(* CODESYS project SLL_IFM_IO_V0.0.1.0_SP16p5.library
   Version: 0.0.1.0
   Title: SLL_IFM_IO
   Placeholder: SLL_IFM_IO
   CompiledLibraryCompatibilityVersion: CODESYS V3.5 SP16 Patch 5
   Company: SLL
   DefaultNamespace: SLL_IFM_IO

Project tree, tasks and I/O mapping:
  libraries: Util, 3.5.15.0 (System); Standard, 3.5.15.0 (System); ifmIOcommon, 2.4.0.0 (ifm electronic); ifmIOconfigDiagProt, 2.0.6.0 (ifm electronic); ifmTypes, 1.9.6.0 (ifm electronic); BASIC, 3.3.3.0 (OSCAT); ifmOutGroup, 2.1.3.0 (ifm electronic); ifmRawCAN, 4.0.3.0 (ifm electronic); ifmDeviceCR07nn, 1.2.2.0 (ifm electronic); SLL_IFM_Version, 0.0.0.2 (SLL)
  Library Information/
    function IsLibReleased [ST]
    function GetLibVersionNumber [ST]
    function GetLibVersion [ST]
  IO/
    data type CRXXXX_OUTPUT_GROUP_PINS
    data type CRXXXX_INPUT_PINS
    CR0709/
      data type CR0709_ALL_INPUTS_DATA
      data type CR0709_ALL_INPUTS_FB
      data type CR0709_ALL_OUTPUTS_DATA
      data type CR0709_ALL_OUTPUTS_FB
      data type CR0709_ALL_OUTPUT_STATES
      Output/
        function CR0709_Get_Output_Pin_Name_Str [ST]
        function CR0709_Get_Output_Pin_Number_Str [ST]
        function CR0709_Get_Output_Pin_Group [ST]
      Input/
        function CR0709_Get_Input_Pin_Number_Str [ST]
        function CR0709_Get_Input_Pin_Name_Str [ST]
      program PLC_CR0709_System [FBD]
    CR721S/
      data type CR721S_ALL_INPUTS_DATA
      data type CR721S_ALL_INPUTS_FB
      data type CR721S_ALL_OUTPUTS_DATA
      data type CR721S_ALL_OUTPUTS_FB
      data type CR721S_ALL_OUTPUT_STATES
    data type CRXXXX_INPUT_DATA
    data type CRXXXX_OUTPUT_DATA
    data type CRXXXX_OUTPUT_STATE_DATA
    FB/
      function block CRXXXX_INPUT_FB [FBD]: Process
      function block CRXXXX_OUTPUT_FB [FBD]: Process
      function block CRXXXX_OUTPUT_GROUP_FB [FBD]: Process
    Input/
      function CR721S_Get_Input_Pin_Number_Str [ST]
      function CR721S_Get_Input_Pin_Name_Str [ST]
      function CR721S_Get_Input_Pin_Connector [ST]
    Output/
      function CR721S_Get_Output_Group_Pin_Number_Str [ST]
      function CR721S_Get_Output_Group_Pin_Name_Str [ST]
      function CR721S_Get_Output_Pin_Name_Str [ST]
      function CR721S_Get_Output_Pin_Number_Str [ST]
      function CR721S_Get_Output_Pin_Group [ST]
      function CR721S_Get_Output_Pin_Connector [ST]
    data type CRXXXX_OUTPUT_PINS
    data type CRXXXX_OUTPUT_GROUP_DATA
    data type CRXXXX_VERSION_DATA
  global variables GVL_IfmIoLibs
  Hardware/
    data type CRXXXX_LINAK_STATUS
    function block Diag_Op_LINAK_Bridge [FBD]
    data type Diag_Op_PWM_Enum
    data type CRXXXX_Freq_Pulse_Readings
    data type Diag_Ip_Signal_Enum
  Func/
    function Get_IFM_DIAG_INFO_STRING [ST]
*)

// IO/CRXXXX_OUTPUT_GROUP_PINS
{attribute 'qualified_only'}
//{attribute 'strict'}
{attribute 'to_string'} 
TYPE CRXXXX_OUTPUT_GROUP_PINS :
(
	GROUP0 :=0000,
	GROUP1 :=0001,
	GROUP2 :=0002,
	GROUP3 :=0003,
	GROUP4 :=0004,
	GROUP5 :=0005
)WORD;
END_TYPE

// IO/CR0709/CR0709_ALL_INPUTS_DATA
TYPE CR0709_ALL_INPUTS_DATA :
STRUCT
	VERSION: DWORD:=16#8000001;	
	IN0100: CRXXXX_INPUT_DATA;
	IN0101: CRXXXX_INPUT_DATA;
	IN0102: CRXXXX_INPUT_DATA;
	IN0103: CRXXXX_INPUT_DATA;
	IN0200: CRXXXX_INPUT_DATA;
	IN0201: CRXXXX_INPUT_DATA;
	IN0202: CRXXXX_INPUT_DATA;
	IN0203: CRXXXX_INPUT_DATA;
	IN0600: CRXXXX_INPUT_DATA;
	IN0601: CRXXXX_INPUT_DATA;
	IN0602: CRXXXX_INPUT_DATA;
	IN0603: CRXXXX_INPUT_DATA;
	IN0700: CRXXXX_INPUT_DATA;
	IN0701: CRXXXX_INPUT_DATA;
	IN0702: CRXXXX_INPUT_DATA;
	IN0703: CRXXXX_INPUT_DATA;
	IN0000: CRXXXX_INPUT_DATA;
	IN0001: CRXXXX_INPUT_DATA;
	IN0002: CRXXXX_INPUT_DATA;
	IN0003: CRXXXX_INPUT_DATA;
	IN0500: CRXXXX_INPUT_DATA;
	IN0501: CRXXXX_INPUT_DATA;
	IN0502: CRXXXX_INPUT_DATA;
	IN0503: CRXXXX_INPUT_DATA;
	IN0400: CRXXXX_INPUT_DATA;
	IN0401: CRXXXX_INPUT_DATA;
	IN0900: CRXXXX_INPUT_DATA;
	IN0901: CRXXXX_INPUT_DATA;
	IN0300: CRXXXX_INPUT_DATA;
	IN0301: CRXXXX_INPUT_DATA;
	IN0800: CRXXXX_INPUT_DATA;
	IN0801: CRXXXX_INPUT_DATA;
END_STRUCT
END_TYPE

// IO/CR0709/CR0709_ALL_INPUTS_FB
TYPE CR0709_ALL_INPUTS_FB :
STRUCT
	VERSION: DWORD:=16#8000001;	
	IN0100: CRXXXX_INPUT_FB;
	IN0101: CRXXXX_INPUT_FB;
	IN0102: CRXXXX_INPUT_FB;
	IN0103: CRXXXX_INPUT_FB;
	IN0200: CRXXXX_INPUT_FB;
	IN0201: CRXXXX_INPUT_FB;
	IN0202: CRXXXX_INPUT_FB;
	IN0203: CRXXXX_INPUT_FB;
	IN0600: CRXXXX_INPUT_FB;
	IN0601: CRXXXX_INPUT_FB;
	IN0602: CRXXXX_INPUT_FB;
	IN0603: CRXXXX_INPUT_FB;
	IN0700: CRXXXX_INPUT_FB;
	IN0701: CRXXXX_INPUT_FB;
	IN0702: CRXXXX_INPUT_FB;
	IN0703: CRXXXX_INPUT_FB;
	IN0000: CRXXXX_INPUT_FB;
	IN0001: CRXXXX_INPUT_FB;
	IN0002: CRXXXX_INPUT_FB;
	IN0003: CRXXXX_INPUT_FB;
	IN0500: CRXXXX_INPUT_FB;
	IN0501: CRXXXX_INPUT_FB;
	IN0502: CRXXXX_INPUT_FB;
	IN0503: CRXXXX_INPUT_FB;
	IN0400: CRXXXX_INPUT_FB;
	IN0401: CRXXXX_INPUT_FB;
	IN0900: CRXXXX_INPUT_FB;
	IN0901: CRXXXX_INPUT_FB;
	IN0300: CRXXXX_INPUT_FB;
	IN0301: CRXXXX_INPUT_FB;
	IN0800: CRXXXX_INPUT_FB;
	IN0801: CRXXXX_INPUT_FB;	
END_STRUCT
END_TYPE

// IO/CRXXXX_INPUT_PINS
{attribute 'qualified_only'}
//{attribute 'strict'}
{attribute 'to_string'}
TYPE CRXXXX_INPUT_PINS :
(
	IN0100:=0100,
	IN0101:=0101,
	IN0102:=0102,
	IN0103:=0103,
	IN0200:=0200,
	IN0201:=0201,
	IN0202:=0202,
	IN0203:=0203,
	IN0600:=0600,
	IN0601:=0601,
	IN0602:=0602,
	IN0603:=0603,
	IN0700:=0700,
	IN0701:=0701,
	IN0702:=0702,
	IN0703:=0703,
	IN0000:=0000,
	IN0001:=0001,
	IN0002:=0002,
	IN0003:=0003,
	IN0500:=0500,
	IN0501:=0501,
	IN0502:=0502,
	IN0503:=0503,
	IN0400:=0400,
	IN0401:=0401,
	IN0900:=0900,
	IN0901:=0901,
	IN0300:=0300,
	IN0301:=0301,
	IN0800:=0800,
	IN0801:=0801,
	
	IN1100:=1100,
	IN1101:=1101,
	IN1102:=1102,
	IN1103:=1103,
	IN1600:=1600,
	IN1601:=1601,
	IN1602:=1602,
	IN1603:=1603,
	
	IN1000:=1000,
	IN1001:=1001,
	IN1002:=1002,
	IN1003:=1003,
	IN1500:=1500,
	IN1501:=1501,
	IN1502:=1502,
	IN1503:=1503,

	IN1200:=1200,
	IN1201:=1201,
	IN1202:=1202,
	IN1203:=1203,
	IN1400:=1400,
	IN1401:=1401,
	IN1402:=1402,
	IN1403:=1403,
	IN1700:=1700,
	IN1701:=1701,
	IN1702:=1702,
	IN1703:=1703,
	IN1800:=1800,
	IN1801:=1801,
	IN1802:=1802,
	IN1803:=1803,
	IN1300:=1300,
	IN1301:=1301,
	IN1302:=1302,
	IN1303:=1303
)WORD;
END_TYPE;

// IO/CR0709/CR0709_ALL_OUTPUTS_DATA
TYPE CR0709_ALL_OUTPUTS_DATA :
STRUCT
	VERSION: DWORD:=16#8000001;	
	OUT0000 : CRXXXX_OUTPUT_DATA;
	OUT0001 : CRXXXX_OUTPUT_DATA;
	OUT0002 : CRXXXX_OUTPUT_DATA;
	OUT0003 : CRXXXX_OUTPUT_DATA;
	OUT0004 : CRXXXX_OUTPUT_DATA;
	OUT0005 : CRXXXX_OUTPUT_DATA;
	OUT0006 : CRXXXX_OUTPUT_DATA;
	OUT0007 : CRXXXX_OUTPUT_DATA;
	OUT0008 : CRXXXX_OUTPUT_DATA;
	OUT0100 : CRXXXX_OUTPUT_DATA;
	OUT0101 : CRXXXX_OUTPUT_DATA;
	OUT0102 : CRXXXX_OUTPUT_DATA;
	OUT0103 : CRXXXX_OUTPUT_DATA;
	OUT0104 : CRXXXX_OUTPUT_DATA;
	OUT0105 : CRXXXX_OUTPUT_DATA;
	OUT0106 : CRXXXX_OUTPUT_DATA;
	OUT0107 : CRXXXX_OUTPUT_DATA;
	OUT0108 : CRXXXX_OUTPUT_DATA;
	OUT0200 : CRXXXX_OUTPUT_DATA;
	OUT0201 : CRXXXX_OUTPUT_DATA;
	OUT0202 : CRXXXX_OUTPUT_DATA;
	OUT0203 : CRXXXX_OUTPUT_DATA;
	OUT0204 : CRXXXX_OUTPUT_DATA;
	OUT0205 : CRXXXX_OUTPUT_DATA;
	OUT0206 : CRXXXX_OUTPUT_DATA;
	OUT0207 : CRXXXX_OUTPUT_DATA;
	OUT0208 : CRXXXX_OUTPUT_DATA;
	OUT3000 : CRXXXX_OUTPUT_DATA;
	OUT3001 : CRXXXX_OUTPUT_DATA;
	
	GROUP0 : CRXXXX_OUTPUT_GROUP_DATA;
	GROUP1 : CRXXXX_OUTPUT_GROUP_DATA;
	GROUP2 : CRXXXX_OUTPUT_GROUP_DATA;
END_STRUCT
END_TYPE

// IO/CR0709/CR0709_ALL_OUTPUTS_FB
TYPE CR0709_ALL_OUTPUTS_FB :
STRUCT
	VERSION: DWORD:=16#8000001;	
	OUT0000 : CRXXXX_OUTPUT_FB;
	OUT0001 : CRXXXX_OUTPUT_FB;
	OUT0002 : CRXXXX_OUTPUT_FB;
	OUT0003 : CRXXXX_OUTPUT_FB;
	OUT0004 : CRXXXX_OUTPUT_FB;
	OUT0005 : CRXXXX_OUTPUT_FB;
	OUT0006 : CRXXXX_OUTPUT_FB;
	OUT0007 : CRXXXX_OUTPUT_FB;
	OUT0008 : CRXXXX_OUTPUT_FB;
	OUT0100 : CRXXXX_OUTPUT_FB;
	OUT0101 : CRXXXX_OUTPUT_FB;
	OUT0102 : CRXXXX_OUTPUT_FB;
	OUT0103 : CRXXXX_OUTPUT_FB;
	OUT0104 : CRXXXX_OUTPUT_FB;
	OUT0105 : CRXXXX_OUTPUT_FB;
	OUT0106 : CRXXXX_OUTPUT_FB;
	OUT0107 : CRXXXX_OUTPUT_FB;
	OUT0108 : CRXXXX_OUTPUT_FB;
	OUT0200 : CRXXXX_OUTPUT_FB;
	OUT0201 : CRXXXX_OUTPUT_FB;
	OUT0202 : CRXXXX_OUTPUT_FB;
	OUT0203 : CRXXXX_OUTPUT_FB;
	OUT0204 : CRXXXX_OUTPUT_FB;
	OUT0205 : CRXXXX_OUTPUT_FB;
	OUT0206 : CRXXXX_OUTPUT_FB;
	OUT0207 : CRXXXX_OUTPUT_FB;
	OUT0208 : CRXXXX_OUTPUT_FB;
	OUT3000 : CRXXXX_OUTPUT_FB;
	OUT3001 : CRXXXX_OUTPUT_FB;
	
	GROUP0 : CRXXXX_OUTPUT_GROUP_FB;
	GROUP1 : CRXXXX_OUTPUT_GROUP_FB;
	GROUP2 : CRXXXX_OUTPUT_GROUP_FB;	
END_STRUCT
END_TYPE

// IO/CR0709/CR0709_ALL_OUTPUT_STATES
TYPE CR0709_ALL_OUTPUT_STATES :
STRUCT
	VERSION: DWORD:=16#8000001;	
	OUT0000 : CRXXXX_OUTPUT_STATE_DATA;
	OUT0001 : CRXXXX_OUTPUT_STATE_DATA;
	OUT0002 : CRXXXX_OUTPUT_STATE_DATA;
	OUT0003 : CRXXXX_OUTPUT_STATE_DATA;
	OUT0004 : CRXXXX_OUTPUT_STATE_DATA;
	OUT0005 : CRXXXX_OUTPUT_STATE_DATA;
	OUT0006 : CRXXXX_OUTPUT_STATE_DATA;
	OUT0007 : CRXXXX_OUTPUT_STATE_DATA;
	OUT0008 : CRXXXX_OUTPUT_STATE_DATA;
	OUT0100 : CRXXXX_OUTPUT_STATE_DATA;
	OUT0101 : CRXXXX_OUTPUT_STATE_DATA;
	OUT0102 : CRXXXX_OUTPUT_STATE_DATA;
	OUT0103 : CRXXXX_OUTPUT_STATE_DATA;
	OUT0104 : CRXXXX_OUTPUT_STATE_DATA;
	OUT0105 : CRXXXX_OUTPUT_STATE_DATA;
	OUT0106 : CRXXXX_OUTPUT_STATE_DATA;
	OUT0107 : CRXXXX_OUTPUT_STATE_DATA;
	OUT0108 : CRXXXX_OUTPUT_STATE_DATA;
	OUT0200 : CRXXXX_OUTPUT_STATE_DATA;
	OUT0201 : CRXXXX_OUTPUT_STATE_DATA;
	OUT0202 : CRXXXX_OUTPUT_STATE_DATA;
	OUT0203 : CRXXXX_OUTPUT_STATE_DATA;
	OUT0204 : CRXXXX_OUTPUT_STATE_DATA;
	OUT0205 : CRXXXX_OUTPUT_STATE_DATA;
	OUT0206 : CRXXXX_OUTPUT_STATE_DATA;
	OUT0207 : CRXXXX_OUTPUT_STATE_DATA;
	OUT0208 : CRXXXX_OUTPUT_STATE_DATA;
	OUT3000 : CRXXXX_OUTPUT_STATE_DATA;
	OUT3001 : CRXXXX_OUTPUT_STATE_DATA;
	
	GROUP0: CRXXXX_OUTPUT_STATE_DATA;
	GROUP1: CRXXXX_OUTPUT_STATE_DATA;
	GROUP2: CRXXXX_OUTPUT_STATE_DATA;	
END_STRUCT
END_TYPE

// IO/CRXXXX_INPUT_DATA
TYPE CRXXXX_INPUT_DATA :
STRUCT
	uiChannel:WORD;
	eMode: ifmIOcommon.MODE_INPUT;
	eFilter: ifmIOcommon.FILTER_INPUT;

	xError:BOOL;
	eDiagInfo:ifmTypes.DIAG_INFO;
	xPrepared:BOOL;
	xValueDigital:BOOL;
	xValueDigital_Prev:BOOL;	
	uiValueAnalogue:UINT;	
	DigitalChanges:WORD;
	
	Signal_Type: Diag_Ip_Signal_Enum;
END_STRUCT
END_TYPE

// IO/CR721S/CR721S_ALL_INPUTS_DATA
TYPE CR721S_ALL_INPUTS_DATA :
STRUCT
	VERSION: DWORD:=16#8000001;	
	IN0100: CRXXXX_INPUT_DATA;
	IN0101: CRXXXX_INPUT_DATA;
	IN0102: CRXXXX_INPUT_DATA;
	IN0103: CRXXXX_INPUT_DATA;
	IN0200: CRXXXX_INPUT_DATA;
	IN0201: CRXXXX_INPUT_DATA;
	IN0202: CRXXXX_INPUT_DATA;
	IN0203: CRXXXX_INPUT_DATA;
	IN0600: CRXXXX_INPUT_DATA;
	IN0601: CRXXXX_INPUT_DATA;
	IN0602: CRXXXX_INPUT_DATA;
	IN0603: CRXXXX_INPUT_DATA;
	IN0700: CRXXXX_INPUT_DATA;
	IN0701: CRXXXX_INPUT_DATA;
	IN0702: CRXXXX_INPUT_DATA;
	IN0703: CRXXXX_INPUT_DATA;
	IN0000: CRXXXX_INPUT_DATA;
	IN0001: CRXXXX_INPUT_DATA;
	IN0002: CRXXXX_INPUT_DATA;
	IN0003: CRXXXX_INPUT_DATA;
	IN0500: CRXXXX_INPUT_DATA;
	IN0501: CRXXXX_INPUT_DATA;
	IN0502: CRXXXX_INPUT_DATA;
	IN0503: CRXXXX_INPUT_DATA;
	IN0400: CRXXXX_INPUT_DATA;
	IN0401: CRXXXX_INPUT_DATA;
	IN0900: CRXXXX_INPUT_DATA;
	IN0901: CRXXXX_INPUT_DATA;
	IN0300: CRXXXX_INPUT_DATA;
	IN0301: CRXXXX_INPUT_DATA;
	IN0800: CRXXXX_INPUT_DATA;
	IN0801: CRXXXX_INPUT_DATA;
	
	IN1100: CRXXXX_INPUT_DATA;
	IN1101: CRXXXX_INPUT_DATA;
	IN1102: CRXXXX_INPUT_DATA;
	IN1103: CRXXXX_INPUT_DATA;
	IN1600: CRXXXX_INPUT_DATA;
	IN1601: CRXXXX_INPUT_DATA;
	IN1602: CRXXXX_INPUT_DATA;
	IN1603: CRXXXX_INPUT_DATA;
	
	IN1000: CRXXXX_INPUT_DATA;
	IN1001: CRXXXX_INPUT_DATA;
	IN1002: CRXXXX_INPUT_DATA;
	IN1003: CRXXXX_INPUT_DATA;
	IN1500: CRXXXX_INPUT_DATA;
	IN1501: CRXXXX_INPUT_DATA;
	IN1502: CRXXXX_INPUT_DATA;
	IN1503: CRXXXX_INPUT_DATA;

	IN1200: CRXXXX_INPUT_DATA;
	IN1201: CRXXXX_INPUT_DATA;
	IN1202: CRXXXX_INPUT_DATA;
	IN1203: CRXXXX_INPUT_DATA;
	IN1400: CRXXXX_INPUT_DATA;
	IN1401: CRXXXX_INPUT_DATA;
	IN1402: CRXXXX_INPUT_DATA;
	IN1403: CRXXXX_INPUT_DATA;
	IN1700: CRXXXX_INPUT_DATA;
	IN1701: CRXXXX_INPUT_DATA;
	IN1702: CRXXXX_INPUT_DATA;
	IN1703: CRXXXX_INPUT_DATA;
	IN1800: CRXXXX_INPUT_DATA;
	IN1801: CRXXXX_INPUT_DATA;
	IN1802: CRXXXX_INPUT_DATA;
	IN1803: CRXXXX_INPUT_DATA;
	IN1300: CRXXXX_INPUT_DATA;
	IN1301: CRXXXX_INPUT_DATA;
	IN1302: CRXXXX_INPUT_DATA;
	IN1303: CRXXXX_INPUT_DATA;
END_STRUCT
END_TYPE

// IO/CRXXXX_OUTPUT_DATA
TYPE CRXXXX_OUTPUT_DATA :
STRUCT
	uiChannel:WORD;
	eMode: ifmIOcommon.MODE_OUTPUT;
	eFilter: ifmIOcommon.FILTER_OUTPUT;	
	uiOpValue: UINT;
	PWM_Flags: Diag_Op_PWM_Enum;
	
	xError:BOOL;
	eDiagInfo:ifmTypes.DIAG_INFO;	
	xPrepared:BOOL;
	xOutState:BOOL;
	uiOutVoltage:UINT;
	uiOutCurrent:UINT;
	
	xGroupError:BOOL;
	xGroupPrepared:BOOL;
	xGroupGroupState:BOOL;
	xGroupValue:BOOL;
END_STRUCT
END_TYPE

// IO/CRXXXX_OUTPUT_STATE_DATA
TYPE CRXXXX_OUTPUT_STATE_DATA :
STRUCT
	uiValue: UINT;
	xReset: BOOL;
	xManAuto: BOOL;
	uiManValue: UINT;
END_STRUCT
END_TYPE

// IO/CR721S/CR721S_ALL_INPUTS_FB
TYPE CR721S_ALL_INPUTS_FB :
STRUCT
	VERSION: DWORD:=16#8000001;	
	IN0100: CRXXXX_INPUT_FB;
	IN0101: CRXXXX_INPUT_FB;
	IN0102: CRXXXX_INPUT_FB;
	IN0103: CRXXXX_INPUT_FB;
	IN0200: CRXXXX_INPUT_FB;
	IN0201: CRXXXX_INPUT_FB;
	IN0202: CRXXXX_INPUT_FB;
	IN0203: CRXXXX_INPUT_FB;
	IN0600: CRXXXX_INPUT_FB;
	IN0601: CRXXXX_INPUT_FB;
	IN0602: CRXXXX_INPUT_FB;
	IN0603: CRXXXX_INPUT_FB;
	IN0700: CRXXXX_INPUT_FB;
	IN0701: CRXXXX_INPUT_FB;
	IN0702: CRXXXX_INPUT_FB;
	IN0703: CRXXXX_INPUT_FB;
	IN0000: CRXXXX_INPUT_FB;
	IN0001: CRXXXX_INPUT_FB;
	IN0002: CRXXXX_INPUT_FB;
	IN0003: CRXXXX_INPUT_FB;
	IN0500: CRXXXX_INPUT_FB;
	IN0501: CRXXXX_INPUT_FB;
	IN0502: CRXXXX_INPUT_FB;
	IN0503: CRXXXX_INPUT_FB;
	IN0400: CRXXXX_INPUT_FB;
	IN0401: CRXXXX_INPUT_FB;
	IN0900: CRXXXX_INPUT_FB;
	IN0901: CRXXXX_INPUT_FB;
	IN0300: CRXXXX_INPUT_FB;
	IN0301: CRXXXX_INPUT_FB;
	IN0800: CRXXXX_INPUT_FB;
	IN0801: CRXXXX_INPUT_FB;
	
	IN1100: CRXXXX_INPUT_FB;
	IN1101: CRXXXX_INPUT_FB;
	IN1102: CRXXXX_INPUT_FB;
	IN1103: CRXXXX_INPUT_FB;
	IN1600: CRXXXX_INPUT_FB;
	IN1601: CRXXXX_INPUT_FB;
	IN1602: CRXXXX_INPUT_FB;
	IN1603: CRXXXX_INPUT_FB;
	
	IN1000: CRXXXX_INPUT_FB;
	IN1001: CRXXXX_INPUT_FB;
	IN1002: CRXXXX_INPUT_FB;
	IN1003: CRXXXX_INPUT_FB;
	IN1500: CRXXXX_INPUT_FB;
	IN1501: CRXXXX_INPUT_FB;
	IN1502: CRXXXX_INPUT_FB;
	IN1503: CRXXXX_INPUT_FB;

	IN1200: CRXXXX_INPUT_FB;
	IN1201: CRXXXX_INPUT_FB;
	IN1202: CRXXXX_INPUT_FB;
	IN1203: CRXXXX_INPUT_FB;
	IN1400: CRXXXX_INPUT_FB;
	IN1401: CRXXXX_INPUT_FB;
	IN1402: CRXXXX_INPUT_FB;
	IN1403: CRXXXX_INPUT_FB;
	IN1700: CRXXXX_INPUT_FB;
	IN1701: CRXXXX_INPUT_FB;
	IN1702: CRXXXX_INPUT_FB;
	IN1703: CRXXXX_INPUT_FB;
	IN1800: CRXXXX_INPUT_FB;
	IN1801: CRXXXX_INPUT_FB;
	IN1802: CRXXXX_INPUT_FB;
	IN1803: CRXXXX_INPUT_FB;
	IN1300: CRXXXX_INPUT_FB;
	IN1301: CRXXXX_INPUT_FB;
	IN1302: CRXXXX_INPUT_FB;
	IN1303: CRXXXX_INPUT_FB;
END_STRUCT
END_TYPE

// IO/CR721S/CR721S_ALL_OUTPUTS_DATA
TYPE CR721S_ALL_OUTPUTS_DATA :
STRUCT
	VERSION: DWORD:=16#8000001;	
	OUT0000 : CRXXXX_OUTPUT_DATA;
	OUT0001 : CRXXXX_OUTPUT_DATA;
	OUT0002 : CRXXXX_OUTPUT_DATA;
	OUT0003 : CRXXXX_OUTPUT_DATA;
	OUT0004 : CRXXXX_OUTPUT_DATA;
	OUT0005 : CRXXXX_OUTPUT_DATA;
	OUT0006 : CRXXXX_OUTPUT_DATA;
	OUT0007 : CRXXXX_OUTPUT_DATA;
	OUT0008 : CRXXXX_OUTPUT_DATA;
	OUT0100 : CRXXXX_OUTPUT_DATA;
	OUT0101 : CRXXXX_OUTPUT_DATA;
	OUT0102 : CRXXXX_OUTPUT_DATA;
	OUT0103 : CRXXXX_OUTPUT_DATA;
	OUT0104 : CRXXXX_OUTPUT_DATA;
	OUT0105 : CRXXXX_OUTPUT_DATA;
	OUT0106 : CRXXXX_OUTPUT_DATA;
	OUT0107 : CRXXXX_OUTPUT_DATA;
	OUT0108 : CRXXXX_OUTPUT_DATA;
	OUT0200 : CRXXXX_OUTPUT_DATA;
	OUT0201 : CRXXXX_OUTPUT_DATA;
	OUT0202 : CRXXXX_OUTPUT_DATA;
	OUT0203 : CRXXXX_OUTPUT_DATA;
	OUT0204 : CRXXXX_OUTPUT_DATA;
	OUT0205 : CRXXXX_OUTPUT_DATA;
	OUT0206 : CRXXXX_OUTPUT_DATA;
	OUT0207 : CRXXXX_OUTPUT_DATA;
	OUT0208 : CRXXXX_OUTPUT_DATA;
	OUT3000 : CRXXXX_OUTPUT_DATA;
	OUT3001 : CRXXXX_OUTPUT_DATA;
	
	OUT0300 : CRXXXX_OUTPUT_DATA;
	OUT0301 : CRXXXX_OUTPUT_DATA;
	OUT0302 : CRXXXX_OUTPUT_DATA;
	OUT0303 : CRXXXX_OUTPUT_DATA;
	OUT0304 : CRXXXX_OUTPUT_DATA;
	OUT0305 : CRXXXX_OUTPUT_DATA;
	OUT0306 : CRXXXX_OUTPUT_DATA;
	OUT0307 : CRXXXX_OUTPUT_DATA;
	OUT0308 : CRXXXX_OUTPUT_DATA;
	OUT0400 : CRXXXX_OUTPUT_DATA;
	OUT0401 : CRXXXX_OUTPUT_DATA;
	OUT0402 : CRXXXX_OUTPUT_DATA;
	OUT0403 : CRXXXX_OUTPUT_DATA;
	OUT0404 : CRXXXX_OUTPUT_DATA;
	OUT0405 : CRXXXX_OUTPUT_DATA;
	OUT0406 : CRXXXX_OUTPUT_DATA;
	OUT0407 : CRXXXX_OUTPUT_DATA;
	OUT0408 : CRXXXX_OUTPUT_DATA;
	OUT0500 : CRXXXX_OUTPUT_DATA;
	OUT0501 : CRXXXX_OUTPUT_DATA;
	OUT0502 : CRXXXX_OUTPUT_DATA;
	OUT0503 : CRXXXX_OUTPUT_DATA;
	OUT0504 : CRXXXX_OUTPUT_DATA;
	OUT0505 : CRXXXX_OUTPUT_DATA;
	OUT0506 : CRXXXX_OUTPUT_DATA;
	OUT0507 : CRXXXX_OUTPUT_DATA;
	OUT0508 : CRXXXX_OUTPUT_DATA;
	OUT3002 : CRXXXX_OUTPUT_DATA;
	
	GROUP0 : CRXXXX_OUTPUT_GROUP_DATA;
	GROUP1 : CRXXXX_OUTPUT_GROUP_DATA;
	GROUP2 : CRXXXX_OUTPUT_GROUP_DATA;
	GROUP3 : CRXXXX_OUTPUT_GROUP_DATA;
	GROUP4 : CRXXXX_OUTPUT_GROUP_DATA;
	GROUP5 : CRXXXX_OUTPUT_GROUP_DATA;	
END_STRUCT
END_TYPE

// IO/CR721S/CR721S_ALL_OUTPUTS_FB
TYPE CR721S_ALL_OUTPUTS_FB :
STRUCT
	VERSION: DWORD:=16#8000001;	
	OUT0000 : CRXXXX_OUTPUT_FB;
	OUT0001 : CRXXXX_OUTPUT_FB;
	OUT0002 : CRXXXX_OUTPUT_FB;
	OUT0003 : CRXXXX_OUTPUT_FB;
	OUT0004 : CRXXXX_OUTPUT_FB;
	OUT0005 : CRXXXX_OUTPUT_FB;
	OUT0006 : CRXXXX_OUTPUT_FB;
	OUT0007 : CRXXXX_OUTPUT_FB;
	OUT0008 : CRXXXX_OUTPUT_FB;
	OUT0100 : CRXXXX_OUTPUT_FB;
	OUT0101 : CRXXXX_OUTPUT_FB;
	OUT0102 : CRXXXX_OUTPUT_FB;
	OUT0103 : CRXXXX_OUTPUT_FB;
	OUT0104 : CRXXXX_OUTPUT_FB;
	OUT0105 : CRXXXX_OUTPUT_FB;
	OUT0106 : CRXXXX_OUTPUT_FB;
	OUT0107 : CRXXXX_OUTPUT_FB;
	OUT0108 : CRXXXX_OUTPUT_FB;
	OUT0200 : CRXXXX_OUTPUT_FB;
	OUT0201 : CRXXXX_OUTPUT_FB;
	OUT0202 : CRXXXX_OUTPUT_FB;
	OUT0203 : CRXXXX_OUTPUT_FB;
	OUT0204 : CRXXXX_OUTPUT_FB;
	OUT0205 : CRXXXX_OUTPUT_FB;
	OUT0206 : CRXXXX_OUTPUT_FB;
	OUT0207 : CRXXXX_OUTPUT_FB;
	OUT0208 : CRXXXX_OUTPUT_FB;
	OUT3000 : CRXXXX_OUTPUT_FB;	
	OUT3001 : CRXXXX_OUTPUT_FB;	
	
	OUT0300 : CRXXXX_OUTPUT_FB;
	OUT0301 : CRXXXX_OUTPUT_FB;
	OUT0302 : CRXXXX_OUTPUT_FB;
	OUT0303 : CRXXXX_OUTPUT_FB;
	OUT0304 : CRXXXX_OUTPUT_FB;
	OUT0305 : CRXXXX_OUTPUT_FB;
	OUT0306 : CRXXXX_OUTPUT_FB;
	OUT0307 : CRXXXX_OUTPUT_FB;
	OUT0308 : CRXXXX_OUTPUT_FB;
	OUT0400 : CRXXXX_OUTPUT_FB;
	OUT0401 : CRXXXX_OUTPUT_FB;
	OUT0402 : CRXXXX_OUTPUT_FB;
	OUT0403 : CRXXXX_OUTPUT_FB;
	OUT0404 : CRXXXX_OUTPUT_FB;
	OUT0405 : CRXXXX_OUTPUT_FB;
	OUT0406 : CRXXXX_OUTPUT_FB;
	OUT0407 : CRXXXX_OUTPUT_FB;
	OUT0408 : CRXXXX_OUTPUT_FB;
	OUT0500 : CRXXXX_OUTPUT_FB;
	OUT0501 : CRXXXX_OUTPUT_FB;
	OUT0502 : CRXXXX_OUTPUT_FB;
	OUT0503 : CRXXXX_OUTPUT_FB;
	OUT0504 : CRXXXX_OUTPUT_FB;
	OUT0505 : CRXXXX_OUTPUT_FB;
	OUT0506 : CRXXXX_OUTPUT_FB;
	OUT0507 : CRXXXX_OUTPUT_FB;
	OUT0508 : CRXXXX_OUTPUT_FB;
	OUT3002 : CRXXXX_OUTPUT_FB;

	GROUP0 : CRXXXX_OUTPUT_GROUP_FB;
	GROUP1 : CRXXXX_OUTPUT_GROUP_FB;
	GROUP2 : CRXXXX_OUTPUT_GROUP_FB;
	GROUP3 : CRXXXX_OUTPUT_GROUP_FB;
	GROUP4 : CRXXXX_OUTPUT_GROUP_FB;
	GROUP5 : CRXXXX_OUTPUT_GROUP_FB;	
END_STRUCT
END_TYPE

// IO/CR721S/CR721S_ALL_OUTPUT_STATES
TYPE CR721S_ALL_OUTPUT_STATES :
STRUCT
	VERSION: DWORD:=16#8000001;	
	OUT0000 : CRXXXX_OUTPUT_STATE_DATA;
	OUT0001 : CRXXXX_OUTPUT_STATE_DATA;
	OUT0002 : CRXXXX_OUTPUT_STATE_DATA;
	OUT0003 : CRXXXX_OUTPUT_STATE_DATA;
	OUT0004 : CRXXXX_OUTPUT_STATE_DATA;
	OUT0005 : CRXXXX_OUTPUT_STATE_DATA;
	OUT0006 : CRXXXX_OUTPUT_STATE_DATA;
	OUT0007 : CRXXXX_OUTPUT_STATE_DATA;
	OUT0008 : CRXXXX_OUTPUT_STATE_DATA;
	OUT0100 : CRXXXX_OUTPUT_STATE_DATA;
	OUT0101 : CRXXXX_OUTPUT_STATE_DATA;
	OUT0102 : CRXXXX_OUTPUT_STATE_DATA;
	OUT0103 : CRXXXX_OUTPUT_STATE_DATA;
	OUT0104 : CRXXXX_OUTPUT_STATE_DATA;
	OUT0105 : CRXXXX_OUTPUT_STATE_DATA;
	OUT0106 : CRXXXX_OUTPUT_STATE_DATA;
	OUT0107 : CRXXXX_OUTPUT_STATE_DATA;
	OUT0108 : CRXXXX_OUTPUT_STATE_DATA;
	OUT0200 : CRXXXX_OUTPUT_STATE_DATA;
	OUT0201 : CRXXXX_OUTPUT_STATE_DATA;
	OUT0202 : CRXXXX_OUTPUT_STATE_DATA;
	OUT0203 : CRXXXX_OUTPUT_STATE_DATA;
	OUT0204 : CRXXXX_OUTPUT_STATE_DATA;
	OUT0205 : CRXXXX_OUTPUT_STATE_DATA;
	OUT0206 : CRXXXX_OUTPUT_STATE_DATA;
	OUT0207 : CRXXXX_OUTPUT_STATE_DATA;
	OUT0208 : CRXXXX_OUTPUT_STATE_DATA;
	OUT3000 : CRXXXX_OUTPUT_STATE_DATA;
	OUT3001 : CRXXXX_OUTPUT_STATE_DATA;

	OUT0300 : CRXXXX_OUTPUT_STATE_DATA;
	OUT0301 : CRXXXX_OUTPUT_STATE_DATA;
	OUT0302 : CRXXXX_OUTPUT_STATE_DATA;
	OUT0303 : CRXXXX_OUTPUT_STATE_DATA;
	OUT0304 : CRXXXX_OUTPUT_STATE_DATA;
	OUT0305 : CRXXXX_OUTPUT_STATE_DATA;
	OUT0306 : CRXXXX_OUTPUT_STATE_DATA;
	OUT0307 : CRXXXX_OUTPUT_STATE_DATA;
	OUT0308 : CRXXXX_OUTPUT_STATE_DATA;
	OUT0400 : CRXXXX_OUTPUT_STATE_DATA;
	OUT0401 : CRXXXX_OUTPUT_STATE_DATA;
	OUT0402 : CRXXXX_OUTPUT_STATE_DATA;
	OUT0403 : CRXXXX_OUTPUT_STATE_DATA;
	OUT0404 : CRXXXX_OUTPUT_STATE_DATA;
	OUT0405 : CRXXXX_OUTPUT_STATE_DATA;
	OUT0406 : CRXXXX_OUTPUT_STATE_DATA;
	OUT0407 : CRXXXX_OUTPUT_STATE_DATA;
	OUT0408 : CRXXXX_OUTPUT_STATE_DATA;
	OUT0500 : CRXXXX_OUTPUT_STATE_DATA;
	OUT0501 : CRXXXX_OUTPUT_STATE_DATA;
	OUT0502 : CRXXXX_OUTPUT_STATE_DATA;
	OUT0503 : CRXXXX_OUTPUT_STATE_DATA;
	OUT0504 : CRXXXX_OUTPUT_STATE_DATA;
	OUT0505 : CRXXXX_OUTPUT_STATE_DATA;
	OUT0506 : CRXXXX_OUTPUT_STATE_DATA;
	OUT0507 : CRXXXX_OUTPUT_STATE_DATA;
	OUT0508 : CRXXXX_OUTPUT_STATE_DATA;
	OUT3002 : CRXXXX_OUTPUT_STATE_DATA;

	GROUP0 : CRXXXX_OUTPUT_STATE_DATA;
	GROUP1 : CRXXXX_OUTPUT_STATE_DATA;
	GROUP2 : CRXXXX_OUTPUT_STATE_DATA;
	GROUP3 : CRXXXX_OUTPUT_STATE_DATA;
	GROUP4 : CRXXXX_OUTPUT_STATE_DATA;
	GROUP5 : CRXXXX_OUTPUT_STATE_DATA;	
END_STRUCT
END_TYPE

// IO/CRXXXX_OUTPUT_PINS
{attribute 'qualified_only'}
//{attribute 'strict'}
{attribute 'to_string'} 
TYPE CRXXXX_OUTPUT_PINS :
(
	OUT0000 :=0000,
	OUT0001 :=0001,
	OUT0002 :=0002,
	OUT0003 :=0003,
	OUT0004 :=0004,
	OUT0005 :=0005,
	OUT0006 :=0006,	
	OUT0007 :=0007,
	OUT0008 :=0008,
	OUT0100 :=0100,
	OUT0101 :=0101,
	OUT0102 :=0102,
	OUT0103 :=0103,
	OUT0104 :=0104,
	OUT0105 :=0105,
	OUT0106 :=0106,
	OUT0107 :=0107,
	OUT0108 :=0108,
	OUT0200 :=0200,
	OUT0201 :=0201,
	OUT0202 :=0202,
	OUT0203 :=0203,
	OUT0204 :=0204,
	OUT0205 :=0205,
	OUT0206 :=0206,
	OUT0207 :=0207,
	OUT0208 :=0208,
	OUT3000 :=3000,
	OUT3001 :=3001,
	
	OUT0300 :=0300,
	OUT0301 :=0301,
	OUT0302 :=0302,
	OUT0303 :=0303,	
	OUT0304 :=0304,
	OUT0305 :=0305,
	OUT0306 :=0306,
	OUT0307 :=0307,
	OUT0308 :=0308,
	OUT0400 :=0400,
	OUT0401 :=0401,
	OUT0402 :=0402,
	OUT0403 :=0403,	
	OUT0404 :=0404,
	OUT0405 :=0405,
	OUT0406 :=0406,
	OUT0407 :=0407,
	OUT0408 :=0408,
	OUT0500 :=0500,
	OUT0501 :=0501,
	OUT0502 :=0502,
	OUT0503 :=0503,	
	OUT0504 :=0504,
	OUT0505 :=0505,
	OUT0506 :=0506,
	OUT0507 :=0507,
	OUT0508 :=0508,
	OUT3002 :=3002	
)WORD;
END_TYPE

// IO/CRXXXX_OUTPUT_GROUP_DATA
TYPE CRXXXX_OUTPUT_GROUP_DATA :
STRUCT
	uiChannel:WORD;
	eMode: ifmOutGroup.MODE_OUTPUT_GROUP;
	eFilter: ifmOutGroup.FILTER_OUTPUT_GROUP;	
	
	xError:BOOL;
	eDiagInfo:ifmTypes.DIAG_INFO;	
	xPrepared:BOOL;
	xGroupState:BOOL;
	uiGroupCurrent:UINT;
	uiVBBxVoltage:UINT;
	uiGroupVoltage:UINT;
	xValue: BOOL;
END_STRUCT
END_TYPE

// IO/CRXXXX_VERSION_DATA
TYPE CRXXXX_VERSION_DATA :
STRUCT
	HEARTBEAT: BOOL;
END_STRUCT
END_TYPE

// Hardware/CRXXXX_LINAK_STATUS
TYPE CRXXXX_LINAK_STATUS :
STRUCT
	xError:BOOL;
	eDiagInfo: ifmTypes.DIAG_INFO;
	xPrepared:	BOOL;
	wOutCurrent: WORD;
	wPosition_FeedbackmV: WORD;
	xDirection:BOOL;
	wPWM:WORD;
END_STRUCT
END_TYPE

// Hardware/Diag_Op_PWM_Enum
{attribute 'qualified_only'}
{attribute 'strict'}
TYPE Diag_Op_PWM_Enum :
(
	PWM_Not_Used := 0,
	PWM_Single_Pin_CSO := 1,
	PWM_Single_Pin_CSI := 2,
	PWM_Bridge_A := 3,
	PWM_Bridge_B := 4
)BYTE;
END_TYPE

// Hardware/CRXXXX_Freq_Pulse_Readings
TYPE CRXXXX_Freq_Pulse_Readings :
STRUCT
	PulseCount:UDINT;
	ValueCycle_us: UDINT;
	Freq: REAL;
	LastUpdate_uS: UDINT;
END_STRUCT
END_TYPE

// Hardware/Diag_Ip_Signal_Enum
{attribute 'qualified_only'}
{attribute 'strict'}
TYPE Diag_Ip_Signal_Enum :
(
	Not_Used := 0,
	Resistance := 1,
	FreqPulseHigh := 2,
	FreqPulseLow := 3,	
	Voltage_0_10v := 4,
	Current_4_20mA := 5
)BYTE;
END_TYPE

// GVL_IfmIoLibs
{attribute 'qualified_only'}
VAR_GLOBAL
END_VAR

// IO/CR0709/Input/CR0709_Get_Input_Pin_Number_Str
FUNCTION CR0709_Get_Input_Pin_Number_Str : STRING
VAR_INPUT
	enum_in: CRXXXX_INPUT_PINS;
END_VAR
VAR
	temp_str:STRING;
END_VAR

CASE enum_in OF
	CRXXXX_INPUT_PINS.IN0100: temp_str:='63';
	CRXXXX_INPUT_PINS.IN0101: temp_str:='64';
	CRXXXX_INPUT_PINS.IN0102: temp_str:='65';
	CRXXXX_INPUT_PINS.IN0103: temp_str:='66';
	CRXXXX_INPUT_PINS.IN0200: temp_str:='67';
	CRXXXX_INPUT_PINS.IN0201: temp_str:='68';
	CRXXXX_INPUT_PINS.IN0202: temp_str:='69';
	CRXXXX_INPUT_PINS.IN0203: temp_str:='70';
	CRXXXX_INPUT_PINS.IN0600: temp_str:='55';
	CRXXXX_INPUT_PINS.IN0601: temp_str:='56';
	CRXXXX_INPUT_PINS.IN0602: temp_str:='57';
	CRXXXX_INPUT_PINS.IN0603: temp_str:='58';
	CRXXXX_INPUT_PINS.IN0700: temp_str:='59';
	CRXXXX_INPUT_PINS.IN0701: temp_str:='60';
	CRXXXX_INPUT_PINS.IN0702: temp_str:='61';
	CRXXXX_INPUT_PINS.IN0703: temp_str:='62';
	
	CRXXXX_INPUT_PINS.IN0000: temp_str:='25';
	CRXXXX_INPUT_PINS.IN0001: temp_str:='26';
	CRXXXX_INPUT_PINS.IN0002: temp_str:='27';
	CRXXXX_INPUT_PINS.IN0003: temp_str:='28';
	CRXXXX_INPUT_PINS.IN0500: temp_str:='40';
	CRXXXX_INPUT_PINS.IN0501: temp_str:='41';
	CRXXXX_INPUT_PINS.IN0502: temp_str:='42';
	CRXXXX_INPUT_PINS.IN0503: temp_str:='43';
	CRXXXX_INPUT_PINS.IN0400: temp_str:='46';
	CRXXXX_INPUT_PINS.IN0401: temp_str:='47';
	CRXXXX_INPUT_PINS.IN0900: temp_str:='38';
	CRXXXX_INPUT_PINS.IN0901: temp_str:='39';
	CRXXXX_INPUT_PINS.IN0300: temp_str:='44';
	CRXXXX_INPUT_PINS.IN0301: temp_str:='45';
	CRXXXX_INPUT_PINS.IN0800: temp_str:='36';
	CRXXXX_INPUT_PINS.IN0801: temp_str:='37';
END_CASE

CR0709_Get_Input_Pin_Number_Str:= CONCAT('p',temp_str);

END_FUNCTION

// IO/CR0709/Input/CR0709_Get_Input_Pin_Name_Str
FUNCTION CR0709_Get_Input_Pin_Name_Str : STRING
VAR_INPUT
	enum_in: CRXXXX_INPUT_PINS;
END_VAR
VAR
	temp_str:STRING;
END_VAR


CR0709_Get_Input_Pin_Name_Str:= TO_STRING(enum_in);

END_FUNCTION

// IO/CR0709/Output/CR0709_Get_Output_Pin_Name_Str
FUNCTION CR0709_Get_Output_Pin_Name_Str : STRING
VAR_INPUT
	enum_in: CRXXXX_OUTPUT_PINS;
END_VAR
VAR
	temp_int:INT;
	temp_str:STRING;
END_VAR

// temp_int:=ANY_TO_INT(enum_in);
// temp_str:=CONCAT('0000',INT_TO_STRING(temp_int));
// temp_str:=Right(temp_str,4);

CR0709_Get_Output_Pin_Name_Str:= TO_STRING(enum_in);

END_FUNCTION

// IO/CR0709/Output/CR0709_Get_Output_Pin_Number_Str
FUNCTION CR0709_Get_Output_Pin_Number_Str : STRING
VAR_INPUT
	enum_in: CRXXXX_OUTPUT_PINS;
END_VAR
VAR
	temp_str:STRING;
END_VAR

CASE enum_in OF
	CRXXXX_OUTPUT_PINS.OUT0000: temp_str:='16';
	CRXXXX_OUTPUT_PINS.OUT0001: temp_str:='17';
	CRXXXX_OUTPUT_PINS.OUT0002: temp_str:='18';
	CRXXXX_OUTPUT_PINS.OUT0003: temp_str:='19';
	CRXXXX_OUTPUT_PINS.OUT0004: temp_str:='20';
	CRXXXX_OUTPUT_PINS.OUT0005: temp_str:='21';
	CRXXXX_OUTPUT_PINS.OUT0006: temp_str:='22';
	CRXXXX_OUTPUT_PINS.OUT0007: temp_str:='23';
	CRXXXX_OUTPUT_PINS.OUT0008: temp_str:='24';
	CRXXXX_OUTPUT_PINS.OUT0100: temp_str:='06';
	CRXXXX_OUTPUT_PINS.OUT0101: temp_str:='07';
	CRXXXX_OUTPUT_PINS.OUT0102: temp_str:='08';
	CRXXXX_OUTPUT_PINS.OUT0103: temp_str:='09';
	CRXXXX_OUTPUT_PINS.OUT0104: temp_str:='10';
	CRXXXX_OUTPUT_PINS.OUT0105: temp_str:='11';
	CRXXXX_OUTPUT_PINS.OUT0106: temp_str:='12';
	CRXXXX_OUTPUT_PINS.OUT0107: temp_str:='13';
	CRXXXX_OUTPUT_PINS.OUT0108: temp_str:='14';
	CRXXXX_OUTPUT_PINS.OUT0200: temp_str:='73';
	CRXXXX_OUTPUT_PINS.OUT0201: temp_str:='74';
	CRXXXX_OUTPUT_PINS.OUT0202: temp_str:='75';
	CRXXXX_OUTPUT_PINS.OUT0203: temp_str:='76';
	CRXXXX_OUTPUT_PINS.OUT0204: temp_str:='77';
	CRXXXX_OUTPUT_PINS.OUT0205: temp_str:='78';
	CRXXXX_OUTPUT_PINS.OUT0206: temp_str:='79';
	CRXXXX_OUTPUT_PINS.OUT0207: temp_str:='80';
	CRXXXX_OUTPUT_PINS.OUT0208: temp_str:='81';
END_CASE

CR0709_Get_Output_Pin_Number_Str:= CONCAT('p',temp_str);

END_FUNCTION

// IO/CR0709/Output/CR0709_Get_Output_Pin_Group
FUNCTION CR0709_Get_Output_Pin_Group : INT
VAR_INPUT
	enum_in: CRXXXX_OUTPUT_PINS;
END_VAR
VAR
	temp_int:INT:=-1;
END_VAR

CASE enum_in OF
	CRXXXX_OUTPUT_PINS.OUT0000,
	CRXXXX_OUTPUT_PINS.OUT0001,
	CRXXXX_OUTPUT_PINS.OUT0002,
	CRXXXX_OUTPUT_PINS.OUT0003,
	CRXXXX_OUTPUT_PINS.OUT0004,
	CRXXXX_OUTPUT_PINS.OUT0005,
	CRXXXX_OUTPUT_PINS.OUT0006,
	CRXXXX_OUTPUT_PINS.OUT0007,
	CRXXXX_OUTPUT_PINS.OUT0008:
		temp_int:=0;

	CRXXXX_OUTPUT_PINS.OUT0100,
	CRXXXX_OUTPUT_PINS.OUT0101,
	CRXXXX_OUTPUT_PINS.OUT0102,
	CRXXXX_OUTPUT_PINS.OUT0103,
	CRXXXX_OUTPUT_PINS.OUT0104,
	CRXXXX_OUTPUT_PINS.OUT0105,
	CRXXXX_OUTPUT_PINS.OUT0106,
	CRXXXX_OUTPUT_PINS.OUT0107,
	CRXXXX_OUTPUT_PINS.OUT0108:
		temp_int:=1;

	CRXXXX_OUTPUT_PINS.OUT0200,
	CRXXXX_OUTPUT_PINS.OUT0201,
	CRXXXX_OUTPUT_PINS.OUT0202,
	CRXXXX_OUTPUT_PINS.OUT0203,
	CRXXXX_OUTPUT_PINS.OUT0204,
	CRXXXX_OUTPUT_PINS.OUT0205,
	CRXXXX_OUTPUT_PINS.OUT0206,
	CRXXXX_OUTPUT_PINS.OUT0207,
	CRXXXX_OUTPUT_PINS.OUT0208:
		temp_int:=2;
END_CASE

CR0709_Get_Output_Pin_Group:= temp_int;

END_FUNCTION

// IO/Output/CR721S_Get_Output_Group_Pin_Number_Str
FUNCTION CR721S_Get_Output_Group_Pin_Number_Str : STRING
VAR_INPUT
	enum_in: CRXXXX_OUTPUT_GROUP_PINS;
END_VAR
VAR
	temp_str:STRING;
END_VAR

CASE enum_in OF
	CRXXXX_OUTPUT_GROUP_PINS.GROUP0: temp_str:='01';
	CRXXXX_OUTPUT_GROUP_PINS.GROUP1: temp_str:='03';
	CRXXXX_OUTPUT_GROUP_PINS.GROUP2: temp_str:='04';
	CRXXXX_OUTPUT_GROUP_PINS.GROUP3: temp_str:='01';
	CRXXXX_OUTPUT_GROUP_PINS.GROUP4: temp_str:='03';
	CRXXXX_OUTPUT_GROUP_PINS.GROUP5: temp_str:='04';
END_CASE

CR721S_Get_Output_Group_Pin_Number_Str:= CONCAT('p',temp_str);

END_FUNCTION

// IO/Output/CR721S_Get_Output_Group_Pin_Name_Str
FUNCTION CR721S_Get_Output_Group_Pin_Name_Str : STRING
VAR_INPUT
	enum_in: CRXXXX_OUTPUT_GROUP_PINS;
END_VAR
VAR
	temp_int:INT;
	temp_str:STRING;
END_VAR

CR721S_Get_Output_Group_Pin_Name_Str:= TO_STRING(enum_in);

END_FUNCTION

// Library Information/IsLibReleased
// This function has been automatically generated from the project information.
FUNCTION IsLibReleased : BOOL
VAR_INPUT
	
END_VAR

IsLibReleased := FALSE;

END_FUNCTION

// Library Information/GetLibVersionNumber
// This function has been automatically generated from the project information.
FUNCTION GetLibVersionNumber : DWORD
VAR_INPUT
	
END_VAR

GetLibVersionNumber := 256;

END_FUNCTION

// Library Information/GetLibVersion
// This function has been automatically generated from the project information.
FUNCTION GetLibVersion : VERSION
VAR_INPUT
	
END_VAR

GetLibVersion.uiMajor := 0;
GetLibVersion.uiMinor := 0;
GetLibVersion.uiServicePack := 1;
GetLibVersion.uiPatch := 0;

END_FUNCTION

// IO/FB/CRXXXX_INPUT_FB
FUNCTION_BLOCK CRXXXX_INPUT_FB
VAR_INPUT
	xResetError:BOOL;
	uiChannel:WORD;
	eMode: ifmIOcommon.MODE_INPUT;
	eFilter: ifmIOcommon.FILTER_INPUT;	
END_VAR
VAR_OUTPUT
END_VAR
VAR
	Input_FB: ifmIOcommon.Input;
	CDL_FB: ifmIOconfigDiagProt.ConfigDiagLevel;
	INIT_CDL: BOOL := FALSE;
END_VAR

VAR_IN_OUT
	IO_CRXXXX_INPUT_DIAG: CRXXXX_INPUT_DATA;
END_VAR

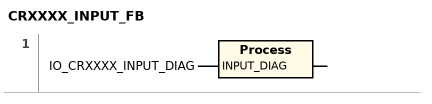
// NETWORK 1
Process(INPUT_DIAG := IO_CRXXXX_INPUT_DIAG);

METHOD PUBLIC Process
VAR_INPUT
END_VAR
VAR_IN_OUT
	INPUT_DIAG: CRXXXX_INPUT_DATA;
END_VAR
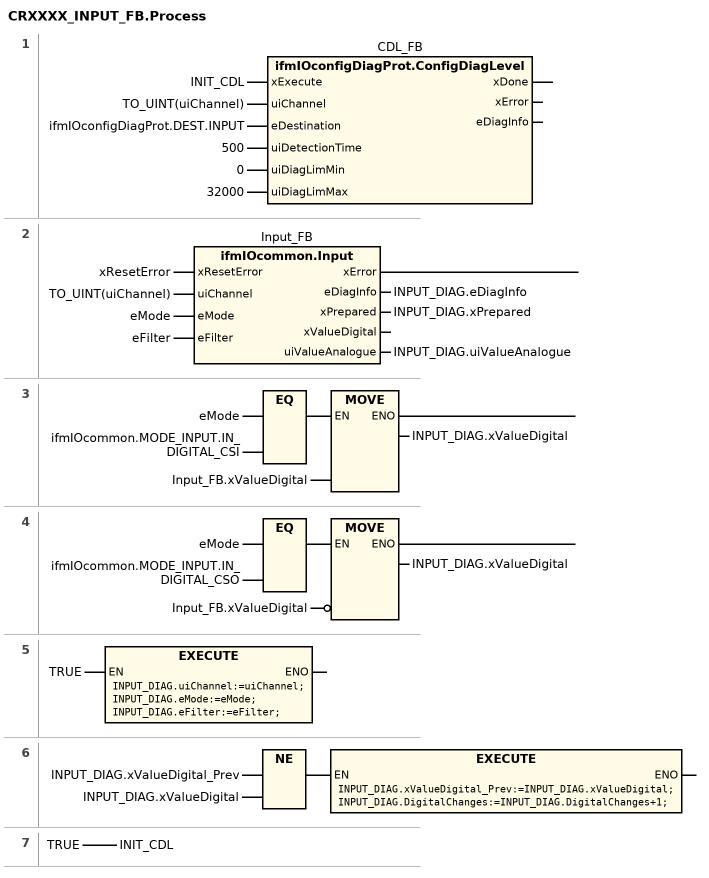
// NETWORK 1
CDL_FB(
    xExecute := INIT_CDL,
    uiChannel := TO_UINT(uiChannel),
    eDestination := ifmIOconfigDiagProt.DEST.INPUT,
    uiDetectionTime := 500,
    uiDiagLimMin := 0,
    uiDiagLimMax := 32000); // ifmIOconfigDiagProt.ConfigDiagLevel

// NETWORK 2
Input_FB(
    xResetError := xResetError,
    uiChannel := TO_UINT(uiChannel),
    eMode := eMode,
    eFilter := eFilter,
    eDiagInfo => INPUT_DIAG.eDiagInfo,
    xPrepared => INPUT_DIAG.xPrepared,
    uiValueAnalogue => INPUT_DIAG.uiValueAnalogue); // ifmIOcommon.Input

// NETWORK 3
IF eMode = ifmIOcommon.MODE_INPUT.IN_DIGITAL_CSI THEN INPUT_DIAG.xValueDigital := Input_FB.xValueDigital; END_IF

// NETWORK 4
IF eMode = ifmIOcommon.MODE_INPUT.IN_DIGITAL_CSO THEN
    INPUT_DIAG.xValueDigital := NOT Input_FB.xValueDigital;
END_IF

// NETWORK 5
INPUT_DIAG.uiChannel:=uiChannel;
INPUT_DIAG.eMode:=eMode;
INPUT_DIAG.eFilter:=eFilter;

// NETWORK 6
IF INPUT_DIAG.xValueDigital_Prev <> INPUT_DIAG.xValueDigital THEN
    INPUT_DIAG.xValueDigital_Prev:=INPUT_DIAG.xValueDigital;
    INPUT_DIAG.DigitalChanges:=INPUT_DIAG.DigitalChanges+1;
END_IF

// NETWORK 7
INIT_CDL := TRUE;
END_METHOD

END_FUNCTION_BLOCK

// IO/FB/CRXXXX_OUTPUT_FB
FUNCTION_BLOCK CRXXXX_OUTPUT_FB
VAR_INPUT
	xResetError:BOOL;
	uiChannel:WORD;
	eMode: ifmIOcommon.MODE_OUTPUT;
	eFilter: ifmIOcommon.FILTER_OUTPUT;
	StateData: CRXXXX_OUTPUT_STATE_DATA;
	Output_Enable: BOOL;
	GRP_OUTPUT_DIAG: REFERENCE TO CRXXXX_OUTPUT_GROUP_DATA;
	CDL_FB: ifmIOconfigDiagProt.ConfigDiagLevel;
	Local_Auto: BOOL:=FALSE;
	Local_uiValue: UINT:=0;
END_VAR
VAR_OUTPUT
END_VAR
VAR
	Output_FB: ifmIOcommon.Output;
END_VAR

VAR_IN_OUT
	IO_CRXXXX_OUTPUT_DIAG: CRXXXX_OUTPUT_DATA;
END_VAR

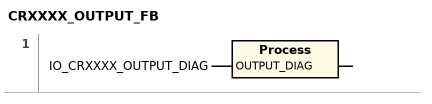
// NETWORK 1
Process(OUTPUT_DIAG := IO_CRXXXX_OUTPUT_DIAG);

METHOD PUBLIC Process
VAR_INPUT
END_VAR

VAR
	uiValue_Prev: UINT;
	uiValue_Changes: UINT;
	INIT_CDL: BOOL:=TRUE;
END_VAR

VAR_IN_OUT
	OUTPUT_DIAG: CRXXXX_OUTPUT_DATA;
END_VAR
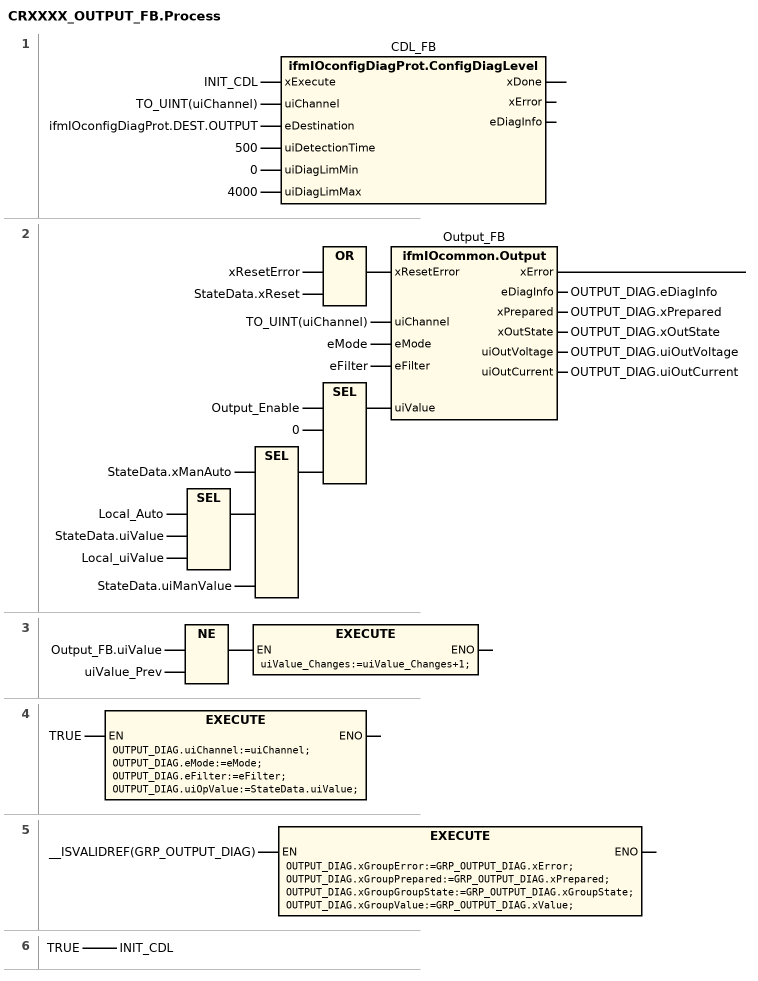
// NETWORK 1
CDL_FB(
    xExecute := INIT_CDL,
    uiChannel := TO_UINT(uiChannel),
    eDestination := ifmIOconfigDiagProt.DEST.OUTPUT,
    uiDetectionTime := 500,
    uiDiagLimMin := 0,
    uiDiagLimMax := 4000); // ifmIOconfigDiagProt.ConfigDiagLevel

// NETWORK 2
Output_FB(
    xResetError := xResetError OR StateData.xReset,
    uiChannel := TO_UINT(uiChannel),
    eMode := eMode,
    eFilter := eFilter,
    uiValue := SEL(Output_Enable, 0, SEL(StateData.xManAuto, SEL(Local_Auto, StateData.uiValue, Local_uiValue), StateData.uiManValue)),
    eDiagInfo => OUTPUT_DIAG.eDiagInfo,
    xPrepared => OUTPUT_DIAG.xPrepared,
    xOutState => OUTPUT_DIAG.xOutState,
    uiOutVoltage => OUTPUT_DIAG.uiOutVoltage,
    uiOutCurrent => OUTPUT_DIAG.uiOutCurrent); // ifmIOcommon.Output

// NETWORK 3
IF Output_FB.uiValue <> uiValue_Prev THEN uiValue_Changes:=uiValue_Changes+1; END_IF

// NETWORK 4
OUTPUT_DIAG.uiChannel:=uiChannel;
OUTPUT_DIAG.eMode:=eMode;
OUTPUT_DIAG.eFilter:=eFilter;
OUTPUT_DIAG.uiOpValue:=StateData.uiValue;

// NETWORK 5
IF __ISVALIDREF(GRP_OUTPUT_DIAG) THEN
    OUTPUT_DIAG.xGroupError:=GRP_OUTPUT_DIAG.xError;
    OUTPUT_DIAG.xGroupPrepared:=GRP_OUTPUT_DIAG.xPrepared;
    OUTPUT_DIAG.xGroupGroupState:=GRP_OUTPUT_DIAG.xGroupState;
    OUTPUT_DIAG.xGroupValue:=GRP_OUTPUT_DIAG.xValue;
END_IF

// NETWORK 6
INIT_CDL := TRUE;
END_METHOD

END_FUNCTION_BLOCK

// IO/Input/CR721S_Get_Input_Pin_Number_Str
FUNCTION CR721S_Get_Input_Pin_Number_Str : STRING
VAR_INPUT
	enum_in: CRXXXX_INPUT_PINS;
END_VAR
VAR
	temp_str:STRING;
END_VAR

CASE enum_in OF
	CRXXXX_INPUT_PINS.IN0100: temp_str:='63';
	CRXXXX_INPUT_PINS.IN0101: temp_str:='64';
	CRXXXX_INPUT_PINS.IN0102: temp_str:='65';
	CRXXXX_INPUT_PINS.IN0103: temp_str:='66';
	CRXXXX_INPUT_PINS.IN0200: temp_str:='67';
	CRXXXX_INPUT_PINS.IN0201: temp_str:='68';
	CRXXXX_INPUT_PINS.IN0202: temp_str:='69';
	CRXXXX_INPUT_PINS.IN0203: temp_str:='70';
	CRXXXX_INPUT_PINS.IN0600: temp_str:='55';
	CRXXXX_INPUT_PINS.IN0601: temp_str:='56';
	CRXXXX_INPUT_PINS.IN0602: temp_str:='57';
	CRXXXX_INPUT_PINS.IN0603: temp_str:='58';
	CRXXXX_INPUT_PINS.IN0700: temp_str:='59';
	CRXXXX_INPUT_PINS.IN0701: temp_str:='60';
	CRXXXX_INPUT_PINS.IN0702: temp_str:='61';
	CRXXXX_INPUT_PINS.IN0703: temp_str:='62';
	
	CRXXXX_INPUT_PINS.IN0000: temp_str:='25';
	CRXXXX_INPUT_PINS.IN0001: temp_str:='26';
	CRXXXX_INPUT_PINS.IN0002: temp_str:='27';
	CRXXXX_INPUT_PINS.IN0003: temp_str:='28';
	CRXXXX_INPUT_PINS.IN0500: temp_str:='40';
	CRXXXX_INPUT_PINS.IN0501: temp_str:='41';
	CRXXXX_INPUT_PINS.IN0502: temp_str:='42';
	CRXXXX_INPUT_PINS.IN0503: temp_str:='43';
	CRXXXX_INPUT_PINS.IN0400: temp_str:='46';
	CRXXXX_INPUT_PINS.IN0401: temp_str:='47';
	CRXXXX_INPUT_PINS.IN0900: temp_str:='38';
	CRXXXX_INPUT_PINS.IN0901: temp_str:='39';
	CRXXXX_INPUT_PINS.IN0300: temp_str:='44';
	CRXXXX_INPUT_PINS.IN0301: temp_str:='45';
	CRXXXX_INPUT_PINS.IN0800: temp_str:='36';
	CRXXXX_INPUT_PINS.IN0801: temp_str:='37';
	
	CRXXXX_INPUT_PINS.IN1100: temp_str:='06';
	CRXXXX_INPUT_PINS.IN1101: temp_str:='07';
	CRXXXX_INPUT_PINS.IN1102: temp_str:='08';
	CRXXXX_INPUT_PINS.IN1103: temp_str:='09';
	CRXXXX_INPUT_PINS.IN1600: temp_str:='36';
	CRXXXX_INPUT_PINS.IN1601: temp_str:='37';
	CRXXXX_INPUT_PINS.IN1602: temp_str:='38';
	CRXXXX_INPUT_PINS.IN1603: temp_str:='39';

	CRXXXX_INPUT_PINS.IN1000: temp_str:='44';
	CRXXXX_INPUT_PINS.IN1001: temp_str:='45';
	CRXXXX_INPUT_PINS.IN1002: temp_str:='46';
	CRXXXX_INPUT_PINS.IN1003: temp_str:='47';
	CRXXXX_INPUT_PINS.IN1500: temp_str:='59';
	CRXXXX_INPUT_PINS.IN1501: temp_str:='60';
	CRXXXX_INPUT_PINS.IN1502: temp_str:='61';
	CRXXXX_INPUT_PINS.IN1503: temp_str:='62';

	CRXXXX_INPUT_PINS.IN1200: temp_str:='10';
	CRXXXX_INPUT_PINS.IN1201: temp_str:='11';
	CRXXXX_INPUT_PINS.IN1202: temp_str:='12';
	CRXXXX_INPUT_PINS.IN1203: temp_str:='13';
	CRXXXX_INPUT_PINS.IN1400: temp_str:='29';
	CRXXXX_INPUT_PINS.IN1401: temp_str:='30';
	CRXXXX_INPUT_PINS.IN1402: temp_str:='31';
	CRXXXX_INPUT_PINS.IN1403: temp_str:='32';
	CRXXXX_INPUT_PINS.IN1700: temp_str:='40';
	CRXXXX_INPUT_PINS.IN1701: temp_str:='41';
	CRXXXX_INPUT_PINS.IN1702: temp_str:='42';
	CRXXXX_INPUT_PINS.IN1703: temp_str:='43';
	CRXXXX_INPUT_PINS.IN1800: temp_str:='55';
	CRXXXX_INPUT_PINS.IN1801: temp_str:='56';
	CRXXXX_INPUT_PINS.IN1802: temp_str:='57';
	CRXXXX_INPUT_PINS.IN1803: temp_str:='58';
	CRXXXX_INPUT_PINS.IN1300: temp_str:='25';
	CRXXXX_INPUT_PINS.IN1301: temp_str:='26';
	CRXXXX_INPUT_PINS.IN1302: temp_str:='27';
	CRXXXX_INPUT_PINS.IN1303: temp_str:='28';
END_CASE

CR721S_Get_Input_Pin_Number_Str:= CONCAT('p',temp_str);

END_FUNCTION

// IO/Input/CR721S_Get_Input_Pin_Name_Str
FUNCTION CR721S_Get_Input_Pin_Name_Str : STRING
VAR_INPUT
	enum_in: CRXXXX_INPUT_PINS;
END_VAR
VAR
	temp_str:STRING;
END_VAR

CR721S_Get_Input_Pin_Name_Str:= TO_STRING(enum_in);

END_FUNCTION

// IO/Output/CR721S_Get_Output_Pin_Name_Str
FUNCTION CR721S_Get_Output_Pin_Name_Str : STRING
VAR_INPUT
	enum_in: CRXXXX_OUTPUT_PINS;
END_VAR
VAR
	temp_int:INT;
	temp_str:STRING;
END_VAR

CR721S_Get_Output_Pin_Name_Str:= TO_STRING(enum_in);

END_FUNCTION

// IO/Output/CR721S_Get_Output_Pin_Number_Str
FUNCTION CR721S_Get_Output_Pin_Number_Str : STRING
VAR_INPUT
	enum_in: CRXXXX_OUTPUT_PINS;
END_VAR
VAR
	temp_str:STRING;
END_VAR

CASE enum_in OF
	CRXXXX_OUTPUT_PINS.OUT0000: temp_str:='16';
	CRXXXX_OUTPUT_PINS.OUT0001: temp_str:='17';
	CRXXXX_OUTPUT_PINS.OUT0002: temp_str:='18';
	CRXXXX_OUTPUT_PINS.OUT0003: temp_str:='19';
	CRXXXX_OUTPUT_PINS.OUT0004: temp_str:='20';
	CRXXXX_OUTPUT_PINS.OUT0005: temp_str:='21';
	CRXXXX_OUTPUT_PINS.OUT0006: temp_str:='22';
	CRXXXX_OUTPUT_PINS.OUT0007: temp_str:='23';
	CRXXXX_OUTPUT_PINS.OUT0008: temp_str:='24';
	CRXXXX_OUTPUT_PINS.OUT0100: temp_str:='06';
	CRXXXX_OUTPUT_PINS.OUT0101: temp_str:='07';
	CRXXXX_OUTPUT_PINS.OUT0102: temp_str:='08';
	CRXXXX_OUTPUT_PINS.OUT0103: temp_str:='09';
	CRXXXX_OUTPUT_PINS.OUT0104: temp_str:='10';
	CRXXXX_OUTPUT_PINS.OUT0105: temp_str:='11';
	CRXXXX_OUTPUT_PINS.OUT0106: temp_str:='12';
	CRXXXX_OUTPUT_PINS.OUT0107: temp_str:='13';
	CRXXXX_OUTPUT_PINS.OUT0108: temp_str:='14';
	CRXXXX_OUTPUT_PINS.OUT0200: temp_str:='73';
	CRXXXX_OUTPUT_PINS.OUT0201: temp_str:='74';
	CRXXXX_OUTPUT_PINS.OUT0202: temp_str:='75';
	CRXXXX_OUTPUT_PINS.OUT0203: temp_str:='76';
	CRXXXX_OUTPUT_PINS.OUT0204: temp_str:='77';
	CRXXXX_OUTPUT_PINS.OUT0205: temp_str:='78';
	CRXXXX_OUTPUT_PINS.OUT0206: temp_str:='79';
	CRXXXX_OUTPUT_PINS.OUT0207: temp_str:='80';
	CRXXXX_OUTPUT_PINS.OUT0208: temp_str:='81';
	CRXXXX_OUTPUT_PINS.OUT3000: temp_str:='31';
	CRXXXX_OUTPUT_PINS.OUT3001: temp_str:='32';	
	
	CRXXXX_OUTPUT_PINS.OUT0300: temp_str:='16';
	CRXXXX_OUTPUT_PINS.OUT0301: temp_str:='17';
	CRXXXX_OUTPUT_PINS.OUT0302: temp_str:='18';
	CRXXXX_OUTPUT_PINS.OUT0303: temp_str:='19';
	CRXXXX_OUTPUT_PINS.OUT0304: temp_str:='20';
	CRXXXX_OUTPUT_PINS.OUT0305: temp_str:='21';
	CRXXXX_OUTPUT_PINS.OUT0306: temp_str:='22';
	CRXXXX_OUTPUT_PINS.OUT0307: temp_str:='23';
	CRXXXX_OUTPUT_PINS.OUT0308: temp_str:='24';
	CRXXXX_OUTPUT_PINS.OUT0400: temp_str:='63';
	CRXXXX_OUTPUT_PINS.OUT0401: temp_str:='64';
	CRXXXX_OUTPUT_PINS.OUT0402: temp_str:='65';
	CRXXXX_OUTPUT_PINS.OUT0403: temp_str:='66';
	CRXXXX_OUTPUT_PINS.OUT0404: temp_str:='67';
	CRXXXX_OUTPUT_PINS.OUT0405: temp_str:='68';
	CRXXXX_OUTPUT_PINS.OUT0406: temp_str:='69';
	CRXXXX_OUTPUT_PINS.OUT0407: temp_str:='70';
	CRXXXX_OUTPUT_PINS.OUT0408: temp_str:='71';
	CRXXXX_OUTPUT_PINS.OUT0500: temp_str:='73';
	CRXXXX_OUTPUT_PINS.OUT0501: temp_str:='74';
	CRXXXX_OUTPUT_PINS.OUT0502: temp_str:='75';
	CRXXXX_OUTPUT_PINS.OUT0503: temp_str:='76';
	CRXXXX_OUTPUT_PINS.OUT0504: temp_str:='77';
	CRXXXX_OUTPUT_PINS.OUT0505: temp_str:='78';
	CRXXXX_OUTPUT_PINS.OUT0506: temp_str:='79';
	CRXXXX_OUTPUT_PINS.OUT0507: temp_str:='80';
	CRXXXX_OUTPUT_PINS.OUT0508: temp_str:='81';
	CRXXXX_OUTPUT_PINS.OUT3002: temp_str:='51';
END_CASE

CR721S_Get_Output_Pin_Number_Str:= CONCAT('p',temp_str);

END_FUNCTION

// IO/Output/CR721S_Get_Output_Pin_Group
FUNCTION CR721S_Get_Output_Pin_Group : INT
VAR_INPUT
	enum_in: CRXXXX_OUTPUT_PINS;
END_VAR
VAR
	temp_int:INT:=-1;
END_VAR

CASE enum_in OF
	CRXXXX_OUTPUT_PINS.OUT0000,
	CRXXXX_OUTPUT_PINS.OUT0001,
	CRXXXX_OUTPUT_PINS.OUT0002,
	CRXXXX_OUTPUT_PINS.OUT0003,
	CRXXXX_OUTPUT_PINS.OUT0004,
	CRXXXX_OUTPUT_PINS.OUT0005,
	CRXXXX_OUTPUT_PINS.OUT0006,
	CRXXXX_OUTPUT_PINS.OUT0007,
	CRXXXX_OUTPUT_PINS.OUT0008:
		temp_int:=0;

	CRXXXX_OUTPUT_PINS.OUT0100,
	CRXXXX_OUTPUT_PINS.OUT0101,
	CRXXXX_OUTPUT_PINS.OUT0102,
	CRXXXX_OUTPUT_PINS.OUT0103,
	CRXXXX_OUTPUT_PINS.OUT0104,
	CRXXXX_OUTPUT_PINS.OUT0105,
	CRXXXX_OUTPUT_PINS.OUT0106,
	CRXXXX_OUTPUT_PINS.OUT0107,
	CRXXXX_OUTPUT_PINS.OUT0108:
		temp_int:=1;

	CRXXXX_OUTPUT_PINS.OUT0200,
	CRXXXX_OUTPUT_PINS.OUT0201,
	CRXXXX_OUTPUT_PINS.OUT0202,
	CRXXXX_OUTPUT_PINS.OUT0203,
	CRXXXX_OUTPUT_PINS.OUT0204,
	CRXXXX_OUTPUT_PINS.OUT0205,
	CRXXXX_OUTPUT_PINS.OUT0206,
	CRXXXX_OUTPUT_PINS.OUT0207,
	CRXXXX_OUTPUT_PINS.OUT0208:
		temp_int:=2;
		
	CRXXXX_OUTPUT_PINS.OUT0300,
	CRXXXX_OUTPUT_PINS.OUT0301,
	CRXXXX_OUTPUT_PINS.OUT0302,
	CRXXXX_OUTPUT_PINS.OUT0303,
	CRXXXX_OUTPUT_PINS.OUT0304,
	CRXXXX_OUTPUT_PINS.OUT0305,
	CRXXXX_OUTPUT_PINS.OUT0306,
	CRXXXX_OUTPUT_PINS.OUT0307,
	CRXXXX_OUTPUT_PINS.OUT0308:
		temp_int:=3;

	CRXXXX_OUTPUT_PINS.OUT0400,
	CRXXXX_OUTPUT_PINS.OUT0401,
	CRXXXX_OUTPUT_PINS.OUT0402,
	CRXXXX_OUTPUT_PINS.OUT0403,
	CRXXXX_OUTPUT_PINS.OUT0404,
	CRXXXX_OUTPUT_PINS.OUT0405,
	CRXXXX_OUTPUT_PINS.OUT0406,
	CRXXXX_OUTPUT_PINS.OUT0407,
	CRXXXX_OUTPUT_PINS.OUT0408:
		temp_int:=4;

	CRXXXX_OUTPUT_PINS.OUT0500,
	CRXXXX_OUTPUT_PINS.OUT0501,
	CRXXXX_OUTPUT_PINS.OUT0502,
	CRXXXX_OUTPUT_PINS.OUT0503,
	CRXXXX_OUTPUT_PINS.OUT0504,
	CRXXXX_OUTPUT_PINS.OUT0505,
	CRXXXX_OUTPUT_PINS.OUT0506,
	CRXXXX_OUTPUT_PINS.OUT0507,
	CRXXXX_OUTPUT_PINS.OUT0508:
		temp_int:=5;		
END_CASE

CR721S_Get_Output_Pin_Group:= temp_int;

END_FUNCTION

// IO/FB/CRXXXX_OUTPUT_GROUP_FB
FUNCTION_BLOCK CRXXXX_OUTPUT_GROUP_FB
VAR_INPUT
	xResetError:BOOL;
	uiChannel:WORD;
	eMode: ifmOutGroup.MODE_OUTPUT_GROUP;
	eFilter: ifmOutGroup.FILTER_OUTPUT_GROUP;
	StateData: CRXXXX_OUTPUT_STATE_DATA;
	Output_Enable: BOOL;
	Local_Auto: BOOL:=FALSE;
	Local_uiValue: UINT:=0;	
END_VAR
VAR_OUTPUT
END_VAR
VAR
	OutputGroup_FB: ifmOutGroup.OutputGroup;	
END_VAR

VAR_IN_OUT
	IO_CRXXXX_OUTPUT_GROUP_DIAG: CRXXXX_OUTPUT_GROUP_DATA;
END_VAR

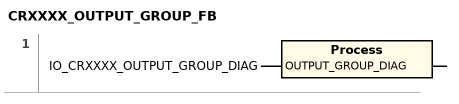
// NETWORK 1
Process(OUTPUT_GROUP_DIAG := IO_CRXXXX_OUTPUT_GROUP_DIAG);

METHOD PUBLIC Process
VAR
END_VAR

VAR_IN_OUT
	OUTPUT_GROUP_DIAG: CRXXXX_OUTPUT_GROUP_DATA;
END_VAR
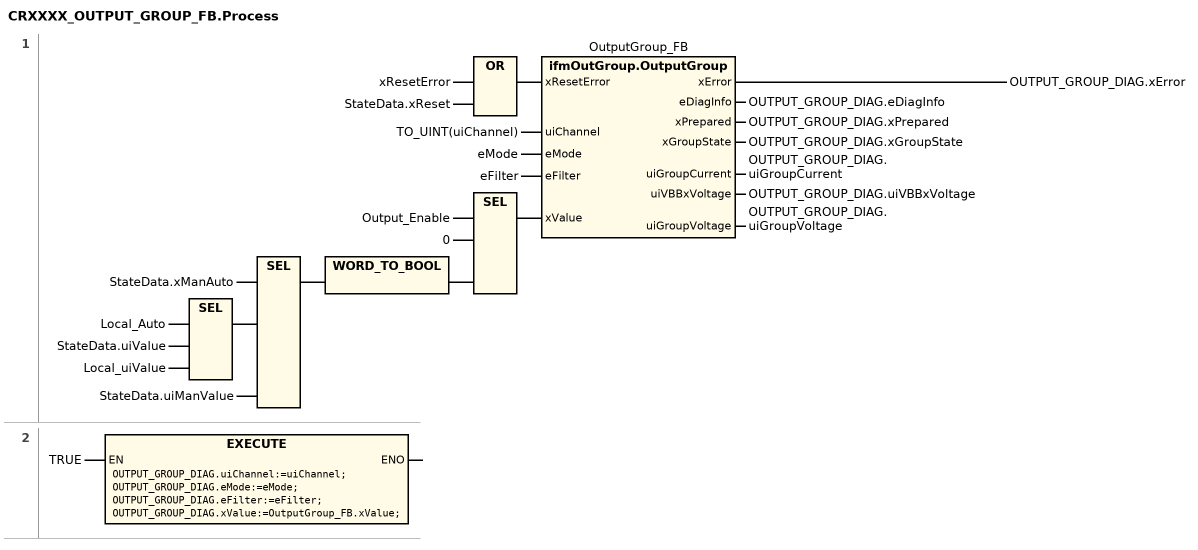
// NETWORK 1
OutputGroup_FB(
    xResetError := xResetError OR StateData.xReset,
    uiChannel := TO_UINT(uiChannel),
    eMode := eMode,
    eFilter := eFilter,
    xValue := SEL(Output_Enable, 0, WORD_TO_BOOL(SEL(StateData.xManAuto, SEL(Local_Auto, StateData.uiValue, Local_uiValue), StateData.uiManValue))),
    eDiagInfo => OUTPUT_GROUP_DIAG.eDiagInfo,
    xPrepared => OUTPUT_GROUP_DIAG.xPrepared,
    xGroupState => OUTPUT_GROUP_DIAG.xGroupState,
    uiGroupCurrent => OUTPUT_GROUP_DIAG.uiGroupCurrent,
    uiVBBxVoltage => OUTPUT_GROUP_DIAG.uiVBBxVoltage,
    uiGroupVoltage => OUTPUT_GROUP_DIAG.uiGroupVoltage); // ifmOutGroup.OutputGroup
OUTPUT_GROUP_DIAG.xError := OutputGroup_FB.xError;

// NETWORK 2
OUTPUT_GROUP_DIAG.uiChannel:=uiChannel;
OUTPUT_GROUP_DIAG.eMode:=eMode;
OUTPUT_GROUP_DIAG.eFilter:=eFilter;
OUTPUT_GROUP_DIAG.xValue:=OutputGroup_FB.xValue;
END_METHOD

END_FUNCTION_BLOCK

// IO/Output/CR721S_Get_Output_Pin_Connector
FUNCTION CR721S_Get_Output_Pin_Connector : INT
VAR_INPUT
	enum_in: CRXXXX_OUTPUT_PINS;
END_VAR
VAR
	temp_int:INT:=-1;
END_VAR

CASE enum_in OF
	CRXXXX_OUTPUT_PINS.OUT0000,
	CRXXXX_OUTPUT_PINS.OUT0001,
	CRXXXX_OUTPUT_PINS.OUT0002,
	CRXXXX_OUTPUT_PINS.OUT0003,
	CRXXXX_OUTPUT_PINS.OUT0004,
	CRXXXX_OUTPUT_PINS.OUT0005,
	CRXXXX_OUTPUT_PINS.OUT0006,
	CRXXXX_OUTPUT_PINS.OUT0007,
	CRXXXX_OUTPUT_PINS.OUT0008,
	CRXXXX_OUTPUT_PINS.OUT0100,
	CRXXXX_OUTPUT_PINS.OUT0101,
	CRXXXX_OUTPUT_PINS.OUT0102,
	CRXXXX_OUTPUT_PINS.OUT0103,
	CRXXXX_OUTPUT_PINS.OUT0104,
	CRXXXX_OUTPUT_PINS.OUT0105,
	CRXXXX_OUTPUT_PINS.OUT0106,
	CRXXXX_OUTPUT_PINS.OUT0107,
	CRXXXX_OUTPUT_PINS.OUT0108,
	CRXXXX_OUTPUT_PINS.OUT0200,
	CRXXXX_OUTPUT_PINS.OUT0201,
	CRXXXX_OUTPUT_PINS.OUT0202,
	CRXXXX_OUTPUT_PINS.OUT0203,
	CRXXXX_OUTPUT_PINS.OUT0204,
	CRXXXX_OUTPUT_PINS.OUT0205,
	CRXXXX_OUTPUT_PINS.OUT0206,
	CRXXXX_OUTPUT_PINS.OUT0207,
	CRXXXX_OUTPUT_PINS.OUT0208:
		temp_int:=0;
		
	CRXXXX_OUTPUT_PINS.OUT0300,
	CRXXXX_OUTPUT_PINS.OUT0301,
	CRXXXX_OUTPUT_PINS.OUT0302,
	CRXXXX_OUTPUT_PINS.OUT0303,
	CRXXXX_OUTPUT_PINS.OUT0304,
	CRXXXX_OUTPUT_PINS.OUT0305,
	CRXXXX_OUTPUT_PINS.OUT0306,
	CRXXXX_OUTPUT_PINS.OUT0307,
	CRXXXX_OUTPUT_PINS.OUT0308,
	CRXXXX_OUTPUT_PINS.OUT0400,
	CRXXXX_OUTPUT_PINS.OUT0401,
	CRXXXX_OUTPUT_PINS.OUT0402,
	CRXXXX_OUTPUT_PINS.OUT0403,
	CRXXXX_OUTPUT_PINS.OUT0404,
	CRXXXX_OUTPUT_PINS.OUT0405,
	CRXXXX_OUTPUT_PINS.OUT0406,
	CRXXXX_OUTPUT_PINS.OUT0407,
	CRXXXX_OUTPUT_PINS.OUT0408,
	CRXXXX_OUTPUT_PINS.OUT0500,
	CRXXXX_OUTPUT_PINS.OUT0501,
	CRXXXX_OUTPUT_PINS.OUT0502,
	CRXXXX_OUTPUT_PINS.OUT0503,
	CRXXXX_OUTPUT_PINS.OUT0504,
	CRXXXX_OUTPUT_PINS.OUT0505,
	CRXXXX_OUTPUT_PINS.OUT0506,
	CRXXXX_OUTPUT_PINS.OUT0507,
	CRXXXX_OUTPUT_PINS.OUT0508:
		temp_int:=1;		
END_CASE

CR721S_Get_Output_Pin_Connector:= temp_int;

END_FUNCTION

// IO/Input/CR721S_Get_Input_Pin_Connector
FUNCTION CR721S_Get_Input_Pin_Connector : INT
VAR_INPUT
	enum_in: CRXXXX_INPUT_PINS;
END_VAR
VAR
	temp_int:INT:=-1;
END_VAR

CASE enum_in OF
	CRXXXX_INPUT_PINS.IN0100,
	CRXXXX_INPUT_PINS.IN0101,
	CRXXXX_INPUT_PINS.IN0102,
	CRXXXX_INPUT_PINS.IN0103,
	CRXXXX_INPUT_PINS.IN0200,
	CRXXXX_INPUT_PINS.IN0201,
	CRXXXX_INPUT_PINS.IN0202,
	CRXXXX_INPUT_PINS.IN0203,
	CRXXXX_INPUT_PINS.IN0600,
	CRXXXX_INPUT_PINS.IN0601,
	CRXXXX_INPUT_PINS.IN0602,
	CRXXXX_INPUT_PINS.IN0603,
	CRXXXX_INPUT_PINS.IN0700,
	CRXXXX_INPUT_PINS.IN0701,
	CRXXXX_INPUT_PINS.IN0702,
	CRXXXX_INPUT_PINS.IN0703,
	CRXXXX_INPUT_PINS.IN0000,
	CRXXXX_INPUT_PINS.IN0001,
	CRXXXX_INPUT_PINS.IN0002,
	CRXXXX_INPUT_PINS.IN0003,
	CRXXXX_INPUT_PINS.IN0500,
	CRXXXX_INPUT_PINS.IN0501,
	CRXXXX_INPUT_PINS.IN0502,
	CRXXXX_INPUT_PINS.IN0503,
	CRXXXX_INPUT_PINS.IN0400,
	CRXXXX_INPUT_PINS.IN0401,
	CRXXXX_INPUT_PINS.IN0900,
	CRXXXX_INPUT_PINS.IN0901,
	CRXXXX_INPUT_PINS.IN0300,
	CRXXXX_INPUT_PINS.IN0301,
	CRXXXX_INPUT_PINS.IN0800,
	CRXXXX_INPUT_PINS.IN0801:
		temp_int:=0;
	
	CRXXXX_INPUT_PINS.IN1100,
	CRXXXX_INPUT_PINS.IN1101,
	CRXXXX_INPUT_PINS.IN1102,
	CRXXXX_INPUT_PINS.IN1103,
	CRXXXX_INPUT_PINS.IN1600,
	CRXXXX_INPUT_PINS.IN1601,
	CRXXXX_INPUT_PINS.IN1602,
	CRXXXX_INPUT_PINS.IN1603,

	CRXXXX_INPUT_PINS.IN1000,
	CRXXXX_INPUT_PINS.IN1001,
	CRXXXX_INPUT_PINS.IN1002,
	CRXXXX_INPUT_PINS.IN1003,
	CRXXXX_INPUT_PINS.IN1500,
	CRXXXX_INPUT_PINS.IN1501,
	CRXXXX_INPUT_PINS.IN1502,
	CRXXXX_INPUT_PINS.IN1503,

	CRXXXX_INPUT_PINS.IN1200,
	CRXXXX_INPUT_PINS.IN1201,
	CRXXXX_INPUT_PINS.IN1202,
	CRXXXX_INPUT_PINS.IN1203,
	CRXXXX_INPUT_PINS.IN1400,
	CRXXXX_INPUT_PINS.IN1401,
	CRXXXX_INPUT_PINS.IN1402,
	CRXXXX_INPUT_PINS.IN1403,
	CRXXXX_INPUT_PINS.IN1700,
	CRXXXX_INPUT_PINS.IN1701,
	CRXXXX_INPUT_PINS.IN1702,
	CRXXXX_INPUT_PINS.IN1703,
	CRXXXX_INPUT_PINS.IN1800,
	CRXXXX_INPUT_PINS.IN1801,
	CRXXXX_INPUT_PINS.IN1802,
	CRXXXX_INPUT_PINS.IN1803,
	CRXXXX_INPUT_PINS.IN1300,
	CRXXXX_INPUT_PINS.IN1301,
	CRXXXX_INPUT_PINS.IN1302,
	CRXXXX_INPUT_PINS.IN1303:
		temp_int:=1;
END_CASE

CR721S_Get_Input_Pin_Connector:= temp_int;

END_FUNCTION

// IO/CR0709/PLC_CR0709_System
PROGRAM PLC_CR0709_System
VAR
	Temperature_PCB_FB: ifmIOcommon.Temperature;
	Temperature_CPU_FB: ifmIOcommon.Temperature;	
	SystemSupply_VBB30_FB: ifmIOcommon.SystemSupply;
	SystemSupply_VBB15_FB: ifmIOcommon.SystemSupply;
	Cycle_Freq_FB: Cycle_Freq_REAL;
	CAN0_Status:  ifmRCAN.CAN_Status;
	CAN1_Status: ifmRCAN.CAN_Status;
	CAN2_Status: ifmRCAN.CAN_Status;
	CAN3_Status: ifmRCAN.CAN_Status;
END_VAR

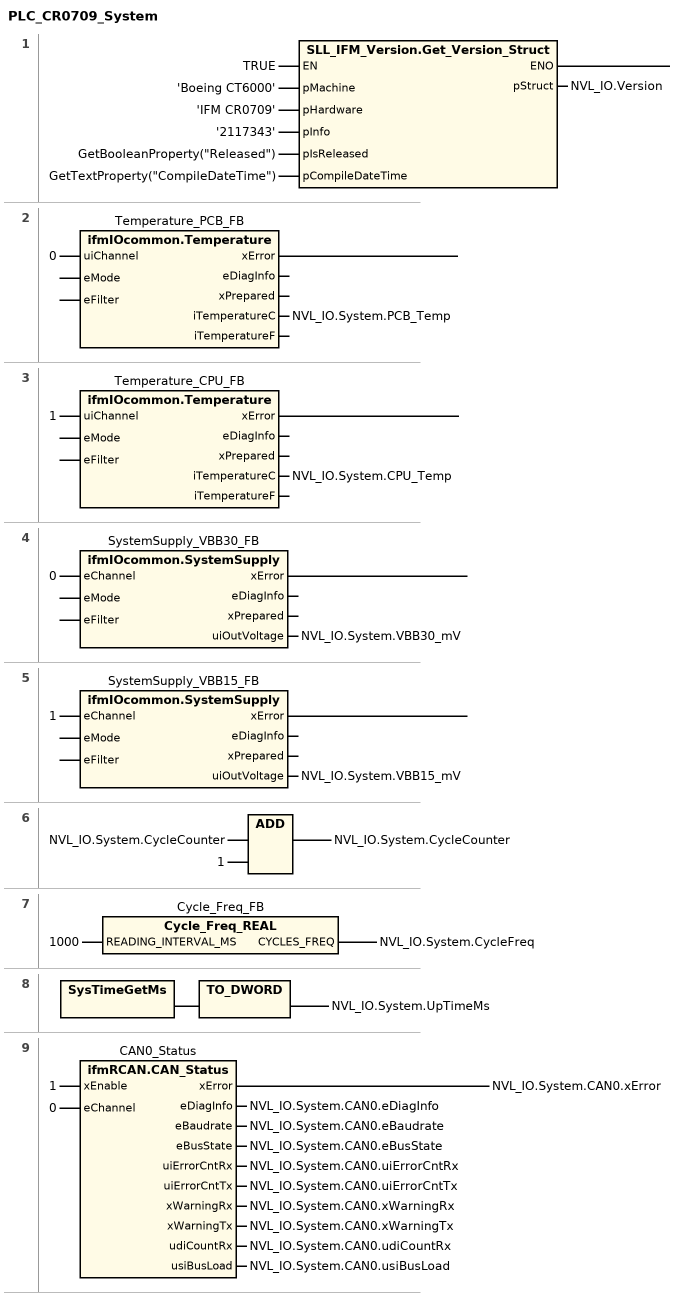
// NETWORK 1
SLL_IFM_Version.Get_Version_Struct(pMachine := 'Boeing CT6000', pHardware := 'IFM CR0709', pInfo := '2117343', pIsReleased := GetBooleanProperty("Released"), pCompileDateTime := GetTextProperty("CompileDateTime"), pStruct => NVL_IO.Version);

// NETWORK 2
Temperature_PCB_FB(uiChannel := 0, iTemperatureC => NVL_IO.System.PCB_Temp); // ifmIOcommon.Temperature

// NETWORK 3
Temperature_CPU_FB(uiChannel := 1, iTemperatureC => NVL_IO.System.CPU_Temp); // ifmIOcommon.Temperature

// NETWORK 4
SystemSupply_VBB30_FB(eChannel := 0, uiOutVoltage => NVL_IO.System.VBB30_mV); // ifmIOcommon.SystemSupply

// NETWORK 5
SystemSupply_VBB15_FB(eChannel := 1, uiOutVoltage => NVL_IO.System.VBB15_mV); // ifmIOcommon.SystemSupply

// NETWORK 6
NVL_IO.System.CycleCounter := NVL_IO.System.CycleCounter + 1;

// NETWORK 7
Cycle_Freq_FB(READING_INTERVAL_MS := 1000); // Cycle_Freq_REAL
NVL_IO.System.CycleFreq := Cycle_Freq_FB.CYCLES_FREQ;

// NETWORK 8
NVL_IO.System.UpTimeMs := TO_DWORD(SysTimeGetMs());

// NETWORK 9
CAN0_Status(
    xEnable := 1,
    eChannel := 0,
    eDiagInfo => NVL_IO.System.CAN0.eDiagInfo,
    eBaudrate => NVL_IO.System.CAN0.eBaudrate,
    eBusState => NVL_IO.System.CAN0.eBusState,
    uiErrorCntRx => NVL_IO.System.CAN0.uiErrorCntRx,
    uiErrorCntTx => NVL_IO.System.CAN0.uiErrorCntTx,
    xWarningRx => NVL_IO.System.CAN0.xWarningRx,
    xWarningTx => NVL_IO.System.CAN0.xWarningTx,
    udiCountRx => NVL_IO.System.CAN0.udiCountRx,
    usiBusLoad => NVL_IO.System.CAN0.usiBusLoad); // ifmRCAN.CAN_Status
NVL_IO.System.CAN0.xError := CAN0_Status.xError;

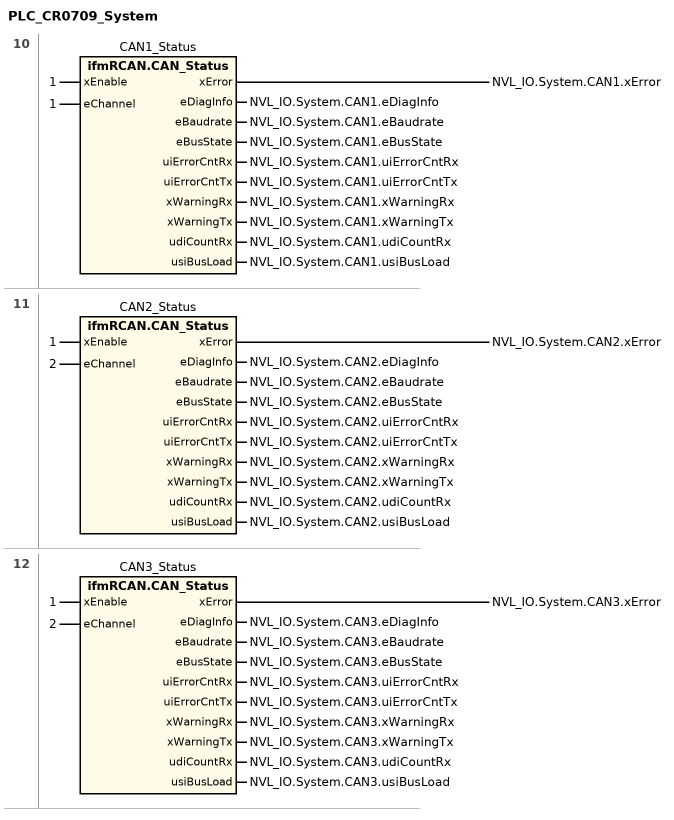
// NETWORK 10
CAN1_Status(
    xEnable := 1,
    eChannel := 1,
    eDiagInfo => NVL_IO.System.CAN1.eDiagInfo,
    eBaudrate => NVL_IO.System.CAN1.eBaudrate,
    eBusState => NVL_IO.System.CAN1.eBusState,
    uiErrorCntRx => NVL_IO.System.CAN1.uiErrorCntRx,
    uiErrorCntTx => NVL_IO.System.CAN1.uiErrorCntTx,
    xWarningRx => NVL_IO.System.CAN1.xWarningRx,
    xWarningTx => NVL_IO.System.CAN1.xWarningTx,
    udiCountRx => NVL_IO.System.CAN1.udiCountRx,
    usiBusLoad => NVL_IO.System.CAN1.usiBusLoad); // ifmRCAN.CAN_Status
NVL_IO.System.CAN1.xError := CAN1_Status.xError;

// NETWORK 11
CAN2_Status(
    xEnable := 1,
    eChannel := 2,
    eDiagInfo => NVL_IO.System.CAN2.eDiagInfo,
    eBaudrate => NVL_IO.System.CAN2.eBaudrate,
    eBusState => NVL_IO.System.CAN2.eBusState,
    uiErrorCntRx => NVL_IO.System.CAN2.uiErrorCntRx,
    uiErrorCntTx => NVL_IO.System.CAN2.uiErrorCntTx,
    xWarningRx => NVL_IO.System.CAN2.xWarningRx,
    xWarningTx => NVL_IO.System.CAN2.xWarningTx,
    udiCountRx => NVL_IO.System.CAN2.udiCountRx,
    usiBusLoad => NVL_IO.System.CAN2.usiBusLoad); // ifmRCAN.CAN_Status
NVL_IO.System.CAN2.xError := CAN2_Status.xError;

// NETWORK 12
CAN3_Status(
    xEnable := 1,
    eChannel := 2,
    eDiagInfo => NVL_IO.System.CAN3.eDiagInfo,
    eBaudrate => NVL_IO.System.CAN3.eBaudrate,
    eBusState => NVL_IO.System.CAN3.eBusState,
    uiErrorCntRx => NVL_IO.System.CAN3.uiErrorCntRx,
    uiErrorCntTx => NVL_IO.System.CAN3.uiErrorCntTx,
    xWarningRx => NVL_IO.System.CAN3.xWarningRx,
    xWarningTx => NVL_IO.System.CAN3.xWarningTx,
    udiCountRx => NVL_IO.System.CAN3.udiCountRx,
    usiBusLoad => NVL_IO.System.CAN3.usiBusLoad); // ifmRCAN.CAN_Status
NVL_IO.System.CAN3.xError := CAN3_Status.xError;

END_PROGRAM

// Hardware/Diag_Op_LINAK_Bridge
FUNCTION_BLOCK Diag_Op_LINAK_Bridge
VAR_INPUT
	CRXXXX_LINAK: CRXXXX_LINAK_STATUS;
END_VAR
VAR_OUTPUT
	OpStringA: STRING;
	OpStringB: STRING;
END_VAR
VAR
END_VAR

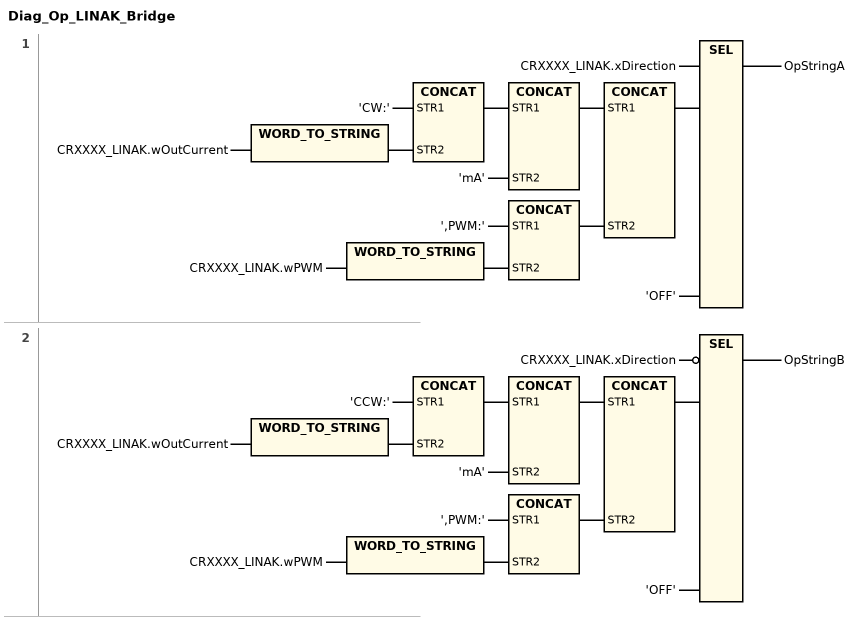
// NETWORK 1
OpStringA := SEL(CRXXXX_LINAK.xDirection, CONCAT(STR1 := CONCAT(STR1 := CONCAT(STR1 := 'CW:', STR2 := WORD_TO_STRING(CRXXXX_LINAK.wOutCurrent)), STR2 := 'mA'), STR2 := CONCAT(STR1 := ',PWM:', STR2 := WORD_TO_STRING(CRXXXX_LINAK.wPWM))), 'OFF');

// NETWORK 2
OpStringB := SEL(NOT CRXXXX_LINAK.xDirection, CONCAT(STR1 := CONCAT(STR1 := CONCAT(STR1 := 'CCW:', STR2 := WORD_TO_STRING(CRXXXX_LINAK.wOutCurrent)), STR2 := 'mA'), STR2 := CONCAT(STR1 := ',PWM:', STR2 := WORD_TO_STRING(CRXXXX_LINAK.wPWM))), 'OFF');

END_FUNCTION_BLOCK

// Func/Get_IFM_DIAG_INFO_STRING
FUNCTION Get_IFM_DIAG_INFO_STRING : STRING
VAR_INPUT
	eDiagInfo:ifmTypes.DIAG_INFO;	
END_VAR
VAR
END_VAR

Get_IFM_DIAG_INFO_STRING:=(TO_STRING(eDiagInfo));

END_FUNCTION
